  // Create log entry
  CreateLogMessagePara1 ( Timestamp   := AxesGroup.State.SystemTime,
                          MessageType := MessageType.CMD,
                          Severity    := Severity.ERROR,
                          MessageCode := ErrorID,
                          MessageText := 'Invalid Parameter ParCmd.JointPosition.E2 = {1}',
                          Para1       := VALID_REAL_TO_STRING(ParCmd.JointPosition.E2));
  RETURN;                          
END_IF


// Check ParCmd.JointPosition.E3 valid ? 
IF ( SysDepIsValidReal(ParCmd.JointPosition.E3) = FALSE ) 
THEN
  // Parameter not valid
  CheckParameterValid := FALSE;
  // Set error
  SetError( ErrorID := RobotLibraryErrorIdEnum.ERR_INVALID_PAR_CMD, Overwrite := TRUE );
  
  // Create log entry
  CreateLogMessagePara1 ( Timestamp   := AxesGroup.State.SystemTime,
                          MessageType := MessageType.CMD,
                          Severity    := Severity.ERROR,
                          MessageCode := ErrorID,
                          MessageText := 'Invalid Parameter ParCmd.JointPosition.E3 = {1}',
                          Para1       := VALID_REAL_TO_STRING(ParCmd.JointPosition.E3));
  RETURN;                          
END_IF


// Check ParCmd.JointPosition.E4 valid ? 
IF ( SysDepIsValidReal(ParCmd.JointPosition.E4) = FALSE ) 
THEN
  // Parameter not valid
  CheckParameterValid := FALSE;
  // Set error
  SetError( ErrorID := RobotLibraryErrorIdEnum.ERR_INVALID_PAR_CMD, Overwrite := TRUE );
  
  // Create log entry
  CreateLogMessagePara1 ( Timestamp   := AxesGroup.State.SystemTime,
                          MessageType := MessageType.CMD,
                          Severity    := Severity.ERROR,
                          MessageCode := ErrorID,
                          MessageText := 'Invalid Parameter ParCmd.JointPosition.E4 = {1}',
                          Para1       := VALID_REAL_TO_STRING(ParCmd.JointPosition.E4));
  RETURN;                          
END_IF


// Check ParCmd.JointPosition.E5 valid ? 
IF ( SysDepIsValidReal(ParCmd.JointPosition.E5) = FALSE ) 
THEN
  // Parameter not valid
  CheckParameterValid := FALSE;
  // Set error
  SetError( ErrorID := RobotLibraryErrorIdEnum.ERR_INVALID_PAR_CMD, Overwrite := TRUE );
  
  // Create log entry
  CreateLogMessagePara1 ( Timestamp   := AxesGroup.State.SystemTime,
                          MessageType := MessageType.CMD,
                          Severity    := Severity.ERROR,
                          MessageCode := ErrorID,
                          MessageText := 'Invalid Parameter ParCmd.JointPosition.E5 = {1}',
                          Para1       := VALID_REAL_TO_STRING(ParCmd.JointPosition.E5));
  RETURN;                          
END_IF


// Check ParCmd.JointPosition.E6 valid ? 
IF ( SysDepIsValidReal(ParCmd.JointPosition.E6) = FALSE ) 
THEN
  // Parameter not valid
  CheckParameterValid := FALSE;
  // Set error
  SetError( ErrorID := RobotLibraryErrorIdEnum.ERR_INVALID_PAR_CMD, Overwrite := TRUE );
  
  // Create log entry
  CreateLogMessagePara1 ( Timestamp   := AxesGroup.State.SystemTime,
                          MessageType := MessageType.CMD,
                          Severity    := Severity.ERROR,
                          MessageCode := ErrorID,
                          MessageText := 'Invalid Parameter ParCmd.JointPosition.E6 = {1}',
                          Para1       := VALID_REAL_TO_STRING(ParCmd.JointPosition.E6));
  RETURN;                          
END_IF


// Check ParCmd.DetectionMode valid ? 
IF (( ParCmd.DetectionMode <> DetectionMode.TORQUE             ) AND
    ( ParCmd.DetectionMode <> DetectionMode.FORCE              ) AND 
    ( ParCmd.DetectionMode <> DetectionMode.ELECTRICAL_CURRENT ) AND 
    ( ParCmd.DetectionMode <> DetectionMode.FOLLOWING_ERROR    ))  
THEN
  // Parameter not valid
  CheckParameterValid := FALSE;
  // Set error
  SetError( ErrorID := RobotLibraryErrorIdEnum.ERR_INVALID_PAR_CMD, Overwrite := TRUE );
  // Create log entry
  CreateLogMessagePara1 ( Timestamp   := AxesGroup.State.SystemTime,
                          MessageType := MessageType.CMD,
                          Severity    := Severity.ERROR,
                          MessageCode := ErrorID,
                          MessageText := 'Invalid Parameter ParCmd.DetectionMode = {1}',
                          Para1       := DETECTION_MODE_TO_STRING(ParCmd.DetectionMode));
  RETURN;                          
END_IF


FOR _idx := 0 TO 6
DO
  // Check ParCmd.DetectionVector[x] valid ? 
  IF ( SysDepIsValidReal(ParCmd.DetectionVector[_idx]) = FALSE ) 
  THEN
    // Parameter not valid
    CheckParameterValid := FALSE;
    // Set error
    SetError( ErrorID := RobotLibraryErrorIdEnum.ERR_INVALID_PAR_CMD, Overwrite := TRUE );
    
    // Create log entry
    CreateLogMessagePara2 ( Timestamp   := AxesGroup.State.SystemTime,
                            MessageType := MessageType.CMD,
                            Severity    := Severity.ERROR,
                            MessageCode := ErrorID,
                            MessageText := 'Invalid Parameter ParCmd.DetectionVector[{2}] = {1}',
                            Para1       := VALID_REAL_TO_STRING(ParCmd.DetectionVector[_idx]),
                            Para2       := DINT_TO_STRING(_idx));
    RETURN;                          
  END_IF
END_FOR


// Check ParCmd.VelocityRate valid ? 
IF  (( SysDepIsValidReal(ParCmd.VelocityRate) = FALSE )  OR
    ((                   ParCmd.VelocityRate  <     0 )  AND 
     (                   ParCmd.VelocityRate <>    -1 )) OR   
     (                   ParCmd.VelocityRate  >   100 ))      
THEN
  // Parameter not valid
  CheckParameterValid := FALSE;
  // Set error
  SetError( ErrorID := RobotLibraryErrorIdEnum.ERR_VELOCITY_INVALID, Overwrite := TRUE );
  // Create log entry
  CreateLogMessagePara1 ( Timestamp   := AxesGroup.State.SystemTime,
                          MessageType := MessageType.CMD,
                          Severity    := Severity.ERROR,
                          MessageCode := ErrorID,
                          MessageText := 'Invalid Parameter ParCmd.VelocityRate = {1}',
                          Para1       := VALID_REAL_TO_STRING(ParCmd.VelocityRate));                            
  RETURN;
END_IF


// Check ParCmd.AccelerationRate valid ? 
IF  (( SysDepIsValidReal(ParCmd.AccelerationRate) = FALSE )  OR
    ((                   ParCmd.AccelerationRate  <     0 )  AND 
     (                   ParCmd.AccelerationRate <>    -1 )) OR   
     (                   ParCmd.AccelerationRate  >   100 ))      
THEN
  // Parameter not valid
  CheckParameterValid := FALSE;
  // Set error
  SetError( ErrorID := RobotLibraryErrorIdEnum.ERR_ACCELERATION_INVALID, Overwrite := TRUE );
  // Create log entry
  CreateLogMessagePara1 ( Timestamp   := AxesGroup.State.SystemTime,
                          MessageType := MessageType.CMD,
                          Severity    := Severity.ERROR,
                          MessageCode := ErrorID,
                          MessageText := 'Invalid Parameter ParCmd.AccelerationRate = {1}',
                          Para1       := VALID_REAL_TO_STRING(ParCmd.AccelerationRate));                            
  RETURN;
END_IF


// Check ParCmd.DecelerationRate valid ? 
IF  (( SysDepIsValidReal(ParCmd.DecelerationRate) = FALSE )  OR
    ((                   ParCmd.DecelerationRate  <     0 )  AND 
     (                   ParCmd.DecelerationRate <>    -1 )) OR   
     (                   ParCmd.DecelerationRate  >   100 ))      
THEN
  // Parameter not valid
  CheckParameterValid := FALSE;
  // Set error
  SetError( ErrorID := RobotLibraryErrorIdEnum.ERR_DECELERATION_INVALID, Overwrite := TRUE );
  // Create log entry
  CreateLogMessagePara1 ( Timestamp   := AxesGroup.State.SystemTime,
                          MessageType := MessageType.CMD,
                          Severity    := Severity.ERROR,
                          MessageCode := ErrorID,
                          MessageText := 'Invalid Parameter ParCmd.DecelerationRate = {1}',
                          Para1       := VALID_REAL_TO_STRING(ParCmd.DecelerationRate));                            
  RETURN;
END_IF


// Check ParCmd.JerkRate valid ? 
IF  (( SysDepIsValidReal(ParCmd.JerkRate) = FALSE )  OR
    ((                   ParCmd.JerkRate  <     0 )  AND 
     (                   ParCmd.JerkRate <>    -1 )) OR   
     (                   ParCmd.JerkRate  >   100 ))      
THEN
  // Parameter not valid
  CheckParameterValid := FALSE;
  // Set error
  SetError( ErrorID := RobotLibraryErrorIdEnum.ERR_JERK_INVALID, Overwrite := TRUE );
  // Create log entry
  CreateLogMessagePara1 ( Timestamp   := AxesGroup.State.SystemTime,
                          MessageType := MessageType.CMD,
                          Severity    := Severity.ERROR,
                          MessageCode := ErrorID,
                          MessageText := 'Invalid Parameter ParCmd.JerkRate = {1}',
                          Para1       := VALID_REAL_TO_STRING(ParCmd.JerkRate));                            
  RETURN;
END_IF


// Check ParCmd.Manipulation
// -> no plausibility check for boolean
                
END_METHOD

METHOD INTERNAL CreateCommandPayload : RobotLibraryCommandDataFB
VAR_IN_OUT
  /// Robot assignment of function
  AxesGroup : AxesGroup; 
END_VAR
VAR
  /// Parameter count
 _parameterCnt : DINT;
END_VAR
// Table 6-412: Sent CMD payload (PLC to RC) of "SearchHardStopJ"
// --------------------------
// Header
// --------------------------
// Byte 00 : UINT  - Type HB     
// Byte 01 :       - Type LB    
// Byte 02 : USINT - Reserve | ExecutionMode
// Byte 03 : USINT - ParSeq  | Priority
// --------------------------
// Datablock
// --------------------------
// Byte 04 : UINT  VelocityRate;
// Byte 05 :       VelocityRate;
// Byte 06 : UINT  AccelerationRate;
// Byte 07 :       AccelerationRate;
// Byte 08 : UINT  DecelerationRate;
// Byte 09 :       DecelerationRate;
// Byte 10 : UINT  JerkRate;
// Byte 11 :       JerkRate;
// Byte 12 : REAL  JointPosition.J1;
// Byte 13 :       JointPosition.J1;
// Byte 14 :       JointPosition.J1;
// Byte 15 :       JointPosition.J1;
// Byte 16 : REAL  JointPosition.J2;
// Byte 17 :       JointPosition.J2;
// Byte 18 :       JointPosition.J2;
// Byte 19 :       JointPosition.J2;
// Byte 20 : REAL  JointPosition.J3;
// Byte 21 :       JointPosition.J3;
// Byte 22 :       JointPosition.J3;
// Byte 23 :       JointPosition.J3;
// Byte 24 : REAL  JointPosition.J4;
// Byte 25 :       JointPosition.J4;
// Byte 26 :       JointPosition.J4;
// Byte 27 :       JointPosition.J4;
// Byte 28 : REAL  JointPosition.J5;
// Byte 29 :       JointPosition.J5;
// Byte 30 :       JointPosition.J5;
// Byte 31 :       JointPosition.J5;
// Byte 32 : REAL  JointPosition.J6;
// Byte 33 :       JointPosition.J6;
// Byte 34 :       JointPosition.J6;
// Byte 35 :       JointPosition.J6;
// Byte 36 : REAL  JointPosition.E1;
// Byte 37 :       JointPosition.E1;
// Byte 38 :       JointPosition.E1;
// Byte 39 :       JointPosition.E1;
// Byte 40 : USINT OriMode;
// Byte 41 : USINT DetectionMode;
// Byte 42 : BOOL  Manipulation;
// Byte 43 : BYTE  Reserved;
// Byte 44 : REAL  DetectionVector[0];
// Byte 45 :       DetectionVector[0];
// Byte 46 :       DetectionVector[0];
// Byte 47 :       DetectionVector[0];
// Byte 48 : REAL  DetectionVector[1];
// Byte 49 :       DetectionVector[1];
// Byte 50 :       DetectionVector[1];
// Byte 51 :       DetectionVector[1];
// Byte 52 : REAL  DetectionVector[2];
// Byte 53 :       DetectionVector[2];
// Byte 54 :       DetectionVector[2];
// Byte 55 :       DetectionVector[2];
// Byte 56 : REAL  DetectionVector[3];
// Byte 57 :       DetectionVector[3];
// Byte 58 :       DetectionVector[3];
// Byte 59 :       DetectionVector[3];
// Byte 60 : REAL  DetectionVector[4];
// Byte 61 :       DetectionVector[4];
// Byte 62 :       DetectionVector[4];
// Byte 63 :       DetectionVector[4];
// Byte 64 : REAL  DetectionVector[5];
// Byte 65 :       DetectionVector[5];
// Byte 66 :       DetectionVector[5];
// Byte 67 :       DetectionVector[5];
// Byte 68 : REAL  JointPosition.E2;
// Byte 69 :       JointPosition.E2;
// Byte 70 :       JointPosition.E2;
// Byte 71 :       JointPosition.E2;
// Byte 72 : REAL  JointPosition.E3;
// Byte 73 :       JointPosition.E3;
// Byte 74 :       JointPosition.E3;
// Byte 75 :       JointPosition.E3;
// Byte 76 : REAL  JointPosition.E4;
// Byte 77 :       JointPosition.E4;
// Byte 78 :       JointPosition.E4;
// Byte 79 :       JointPosition.E4;
// Byte 80 : REAL  JointPosition.E5;
// Byte 81 :       JointPosition.E5;
// Byte 82 :       JointPosition.E5;
// Byte 83 :       JointPosition.E5;
// Byte 84 : REAL  JointPosition.E6;
// Byte 85 :       JointPosition.E6;
// Byte 86 :       JointPosition.E6;
// Byte 87 :       JointPosition.E6;
// --------------------------
                  // set command parameter 
_command.CmdTyp            :=  CmdType.SearchHardstopJ;
_command.ExecMode          :=  ExecMode;
_command.ParSeq            := _command.ParSeq;
_command.Priority          :=  Priority;
_command.VelocityRate      :=  REAL_TO_PERCENT_UINT(_parCmd.VelocityRate     , IsOptional := FALSE);
_command.AccelerationRate  :=  REAL_TO_PERCENT_UINT(_parCmd.AccelerationRate , IsOptional := FALSE);
_command.DecelerationRate  :=  REAL_TO_PERCENT_UINT(_parCmd.DecelerationRate , IsOptional := TRUE );
_command.JerkRate          :=  REAL_TO_PERCENT_UINT(_parCmd.JerkRate         , IsOptional := TRUE );
_command.JointPosition     := _parCmd.JointPosition;
_command.OriMode           := 0;
_command.DetectionMode     := _parCmd.DetectionMode;
_command.Manipulation      := _parCmd.Manipulation;
_command.Reserve           :=  0;
_command.DetectionVector   := _parCmd.DetectionVector;

// copy command data to header
_cmdHeader := _command;
// call base implementation to copy header to payload buffer
CreateCommandPayload := SUPER^.CreateCommandPayload(AxesGroup := AxesGroup);


// Check parameter must be added ? 
IF ( CheckAddParameter(CreateCommandPayload.PayloadPtr))
THEN
  // add command.VelocityRate
  CreateCommandPayload.AddUint(_command.VelocityRate);
  // inc parameter counter
 _parameterCnt := _parameterCnt + 1;  
END_IF

// Check parameter must be added ? 
IF ( CheckAddParameter(CreateCommandPayload.PayloadPtr))
THEN
  // add command.AccelerationRate
  CreateCommandPayload.AddUint(_command.AccelerationRate);
  // inc parameter counter
 _parameterCnt := _parameterCnt + 1;  
END_IF


// Check parameter must be added ? 
IF ( CheckAddParameter(CreateCommandPayload.PayloadPtr))
THEN
  // add command.DecelerationRate
  CreateCommandPayload.AddUint(_command.DecelerationRate);
  // inc parameter counter
 _parameterCnt := _parameterCnt + 1;  
END_IF


// Check parameter must be added ? 
IF ( CheckAddParameter(CreateCommandPayload.PayloadPtr))
THEN
  // add command.JerkRate
  CreateCommandPayload.AddUint(_command.JerkRate);
  // inc parameter counter
 _parameterCnt := _parameterCnt + 1;  
END_IF


// Check parameter must be added ? 
IF ( CheckAddParameter(CreateCommandPayload.PayloadPtr))
THEN
  // add command.JointPosition.J1
  CreateCommandPayload.AddReal(_command.JointPosition.J1);
  // inc parameter counter
 _parameterCnt := _parameterCnt + 1;  
END_IF


// Check parameter must be added ? 
IF ( CheckAddParameter(CreateCommandPayload.PayloadPtr))
THEN
  // add command.JointPosition.J2
  CreateCommandPayload.AddReal(_command.JointPosition.J2);
  // inc parameter counter
 _parameterCnt := _parameterCnt + 1;  
END_IF


// Check parameter must be added ? 
IF ( CheckAddParameter(CreateCommandPayload.PayloadPtr))
THEN
  // add command.JointPosition.J3
  CreateCommandPayload.AddReal(_command.JointPosition.J3);
  // inc parameter counter
 _parameterCnt := _parameterCnt + 1;  
END_IF


// Check parameter must be added ? 
IF ( CheckAddParameter(CreateCommandPayload.PayloadPtr))
THEN
  // add command.JointPosition.J4
  CreateCommandPayload.AddReal(_command.JointPosition.J4);
  // inc parameter counter
 _parameterCnt := _parameterCnt + 1;  
END_IF


// Check parameter must be added ? 
IF ( CheckAddParameter(CreateCommandPayload.PayloadPtr))
THEN
  // add command.JointPosition.J5
  CreateCommandPayload.AddReal(_command.JointPosition.J5);
  // inc parameter counter
 _parameterCnt := _parameterCnt + 1;  
END_IF


// Check parameter must be added ? 
IF ( CheckAddParameter(CreateCommandPayload.PayloadPtr))
THEN
  // add command.JointPosition.J6
  CreateCommandPayload.AddReal(_command.JointPosition.J6);
  // inc parameter counter
 _parameterCnt := _parameterCnt + 1;  
END_IF


// Check parameter must be added ? 
IF ( CheckAddParameter(CreateCommandPayload.PayloadPtr))
THEN
  // add command.JointPosition.E1
  CreateCommandPayload.AddReal(_command.JointPosition.E1);
  // inc parameter counter
 _parameterCnt := _parameterCnt + 1;  
END_IF


// Check parameter must be added ? 
IF ( CheckAddParameter(CreateCommandPayload.PayloadPtr))
THEN
  // add command.OriMode
  CreateCommandPayload.AddUsint(_command.OriMode);
  // inc parameter counter
 _parameterCnt := _parameterCnt + 1;  
END_IF


// Check parameter must be added ? 
IF ( CheckAddParameter(CreateCommandPayload.PayloadPtr))
THEN
  // add command.DetectionMode
  CreateCommandPayload.AddUsint(_command.DetectionMode);
  // inc parameter counter
 _parameterCnt := _parameterCnt + 1;  
END_IF


// Check parameter must be added ? 
IF ( CheckAddParameter(CreateCommandPayload.PayloadPtr))
THEN
  // add command.Manipulation
  CreateCommandPayload.AddBool(_command.Manipulation);
  // inc parameter counter
 _parameterCnt := _parameterCnt + 1;  
END_IF


// Check parameter must be added ? 
IF ( CheckAddParameter(CreateCommandPayload.PayloadPtr))
THEN
  // add command.Reserve
  CreateCommandPayload.AddByte(_command.Reserve);
  // inc parameter counter
 _parameterCnt := _parameterCnt + 1;  
END_IF


// Check parameter must be added ? 
IF ( CheckAddParameter(CreateCommandPayload.PayloadPtr))
THEN
  // add command.DetectionVector[0]
  CreateCommandPayload.AddReal(_command.DetectionVector[0]);
  // inc parameter counter
 _parameterCnt := _parameterCnt + 1;  
END_IF


// Check parameter must be added ? 
IF ( CheckAddParameter(CreateCommandPayload.PayloadPtr))
THEN
  // add command.DetectionVector[1]
  CreateCommandPayload.AddReal(_command.DetectionVector[1]);
  // inc parameter counter
 _parameterCnt := _parameterCnt + 1;  
END_IF


// Check parameter must be added ? 
IF ( CheckAddParameter(CreateCommandPayload.PayloadPtr))
THEN
  // add command.DetectionVector[2]
  CreateCommandPayload.AddReal(_command.DetectionVector[2]);
  // inc parameter counter
 _parameterCnt := _parameterCnt + 1;  
END_IF


// Check parameter must be added ? 
IF ( CheckAddParameter(CreateCommandPayload.PayloadPtr))
THEN
  // add command.DetectionVector[3]
  CreateCommandPayload.AddReal(_command.DetectionVector[3]);
  // inc parameter counter
 _parameterCnt := _parameterCnt + 1;  
END_IF


// Check parameter must be added ? 
IF ( CheckAddParameter(CreateCommandPayload.PayloadPtr))
THEN
  // add command.DetectionVector[4]
  CreateCommandPayload.AddReal(_command.DetectionVector[4]);
  // inc parameter counter
 _parameterCnt := _parameterCnt + 1;  
END_IF


// Check parameter must be added ? 
IF ( CheckAddParameter(CreateCommandPayload.PayloadPtr))
THEN
  // add command.DetectionVector[5]
  CreateCommandPayload.AddReal(_command.DetectionVector[5]);
  // inc parameter counter
 _parameterCnt := _parameterCnt + 1;  
END_IF


// Check parameter must be added ? 
IF ( CheckAddParameter(CreateCommandPayload.PayloadPtr))
THEN
  // add command.JointPosition.E2
  CreateCommandPayload.AddReal(_command.JointPosition.E2);
  // inc parameter counter
 _parameterCnt := _parameterCnt + 1;  
END_IF


// Check parameter must be added ? 
IF ( CheckAddParameter(CreateCommandPayload.PayloadPtr))
THEN
  // add command.JointPosition.E3
  CreateCommandPayload.AddReal(_command.JointPosition.E3);
  // inc parameter counter
 _parameterCnt := _parameterCnt + 1;  
END_IF


// Check parameter must be added ? 
IF ( CheckAddParameter(CreateCommandPayload.PayloadPtr))
THEN
  // add command.JointPosition.E4
  CreateCommandPayload.AddReal(_command.JointPosition.E4);
  // inc parameter counter
 _parameterCnt := _parameterCnt + 1;  
END_IF


// Check parameter must be added ? 
IF ( CheckAddParameter(CreateCommandPayload.PayloadPtr))
THEN
  // add command.JointPosition.E5
  CreateCommandPayload.AddReal(_command.JointPosition.E5);
  // inc parameter counter
 _parameterCnt := _parameterCnt + 1;  
END_IF


// Check parameter must be added ? 
IF ( CheckAddParameter(CreateCommandPayload.PayloadPtr))
THEN
  // add command.JointPosition.E6
  CreateCommandPayload.AddReal(_command.JointPosition.E6);
  // inc parameter counter
 _parameterCnt := _parameterCnt + 1;  
END_IF

  
// Create logging
CreateCommandPayloadLog(AxesGroup := AxesGroup, ParameterCnt := _parameterCnt);
                
END_METHOD

METHOD INTERNAL CreateCommandPayloadLog
VAR_IN_OUT
  /// Robot assignment of function
  AxesGroup : AxesGroup; 
END_VAR
VAR_INPUT
  /// Parameter count
  ParameterCnt : DINT;
END_VAR
VAR 
  /// internal index for loops
 _idx : DINT;
END_VAR
                  // Create log entry for Parameter start
CreateLogMessagePara1 ( Timestamp   := AxesGroup.State.SystemTime,
                        MessageType := MessageType.CMD,
                        Severity    := Severity.DEBUG,
                        MessageCode := 0,
                        MessageText := 'Create command payload with {1} parameter(s) :',
                        Para1       := DINT_TO_STRING(ParameterCnt));
  

// Return if no parameter is remaining...
IF ( ParameterCnt = 0 ) THEN RETURN; END_IF
// dec remaining parameter(s)                        
ParameterCnt := ParameterCnt - 1;
// Create log entry for VelocityRate
CreateLogMessagePara1 ( Timestamp   := AxesGroup.State.SystemTime,
                        MessageType := MessageType.CMD,
                        Severity    := Severity.DEBUG,
                        MessageCode := 0,
                        MessageText := 'Command.VelocityRate = {1}',
                        Para1       :=  UINT_TO_STRING(_command.VelocityRate));


// Return if no parameter is remaining...
IF ( ParameterCnt = 0 ) THEN RETURN; END_IF
// dec remaining parameter(s)                        
ParameterCnt := ParameterCnt - 1;
// Create log entry for AccelerationRate
CreateLogMessagePara1 ( Timestamp   := AxesGroup.State.SystemTime,
                        MessageType := MessageType.CMD,
                        Severity    := Severity.DEBUG,
                        MessageCode := 0,
                        MessageText := 'Command.AccelerationRate = {1}',
                        Para1       :=  UINT_TO_STRING(_command.AccelerationRate));
                        

// Return if no parameter is remaining...
IF ( ParameterCnt = 0 ) THEN RETURN; END_IF
// dec remaining parameter(s)                        
ParameterCnt := ParameterCnt - 1;
// Create log entry for DecelerationRate
CreateLogMessagePara1 ( Timestamp   := AxesGroup.State.SystemTime,
                        MessageType := MessageType.CMD,
                        Severity    := Severity.DEBUG,
                        MessageCode := 0,
                        MessageText := 'Command.DecelerationRate = {1}',
                        Para1       :=  UINT_TO_STRING(_command.DecelerationRate));


// Return if no parameter is remaining...
IF ( ParameterCnt = 0 ) THEN RETURN; END_IF
// dec remaining parameter(s)                        
ParameterCnt := ParameterCnt - 1;
// Create log entry for JerkRate
CreateLogMessagePara1 ( Timestamp   := AxesGroup.State.SystemTime,
                        MessageType := MessageType.CMD,
                        Severity    := Severity.DEBUG,
                        MessageCode := 0,
                        MessageText := 'Command.JerkRate = {1}',
                        Para1       :=  UINT_TO_STRING(_command.JerkRate));


// Return if no parameter is remaining...
IF ( ParameterCnt = 0 ) THEN RETURN; END_IF
// dec remaining parameter(s)                        
ParameterCnt := ParameterCnt - 1;
// Create log entry for JointPosition.J1
CreateLogMessagePara1 ( Timestamp   := AxesGroup.State.SystemTime,
                        MessageType := MessageType.CMD,
                        Severity    := Severity.DEBUG,
                        MessageCode := 0,
                        MessageText := 'Command.JointPosition.J1 = {1}',
                        Para1       :=  REAL_TO_STRING(_command.JointPosition.J1));


// Return if no parameter is remaining...
IF ( ParameterCnt = 0 ) THEN RETURN; END_IF
// dec remaining parameter(s)                        
ParameterCnt := ParameterCnt - 1;
// Create log entry for JointPosition.J2
CreateLogMessagePara1 ( Timestamp   := AxesGroup.State.SystemTime,
                        MessageType := MessageType.CMD,
                        Severity    := Severity.DEBUG,
                        MessageCode := 0,
                        MessageText := 'Command.JointPosition.J2 = {1}',
                        Para1       :=  REAL_TO_STRING(_command.JointPosition.J2));


// Return if no parameter is remaining...
IF ( ParameterCnt = 0 ) THEN RETURN; END_IF
// dec remaining parameter(s)                        
ParameterCnt := ParameterCnt - 1;
// Create log entry for JointPosition.J3
CreateLogMessagePara1 ( Timestamp   := AxesGroup.State.SystemTime,
                        MessageType := MessageType.CMD,
                        Severity    := Severity.DEBUG,
                        MessageCode := 0,
                        MessageText := 'Command.JointPosition.J3 = {1}',
                        Para1       :=  REAL_TO_STRING(_command.JointPosition.J3));


// Return if no parameter is remaining...
IF ( ParameterCnt = 0 ) THEN RETURN; END_IF
// dec remaining parameter(s)                        
ParameterCnt := ParameterCnt - 1;
// Create log entry for JointPosition.J4
CreateLogMessagePara1 ( Timestamp   := AxesGroup.State.SystemTime,
                        MessageType := MessageType.CMD,
                        Severity    := Severity.DEBUG,
                        MessageCode := 0,
                        MessageText := 'Command.JointPosition.J4 = {1}',
                        Para1       :=  REAL_TO_STRING(_command.JointPosition.J4));


// Return if no parameter is remaining...
IF ( ParameterCnt = 0 ) THEN RETURN; END_IF
// dec remaining parameter(s)                        
ParameterCnt := ParameterCnt - 1;
// Create log entry for JointPosition.J5
CreateLogMessagePara1 ( Timestamp   := AxesGroup.State.SystemTime,
                        MessageType := MessageType.CMD,
                        Severity    := Severity.DEBUG,
                        MessageCode := 0,
                        MessageText := 'Command.JointPosition.J5 = {1}',
                        Para1       :=  REAL_TO_STRING(_command.JointPosition.J5));


// Return if no parameter is remaining...
IF ( ParameterCnt = 0 ) THEN RETURN; END_IF
// dec remaining parameter(s)                        
ParameterCnt := ParameterCnt - 1;
// Create log entry for JointPosition.J6
CreateLogMessagePara1 ( Timestamp   := AxesGroup.State.SystemTime,
                        MessageType := MessageType.CMD,
                        Severity    := Severity.DEBUG,
                        MessageCode := 0,
                        MessageText := 'Command.JointPosition.J6 = {1}',
                        Para1       :=  REAL_TO_STRING(_command.JointPosition.J6));


// Return if no parameter is remaining...
IF ( ParameterCnt = 0 ) THEN RETURN; END_IF
// dec remaining parameter(s)                        
ParameterCnt := ParameterCnt - 1;
// Create log entry for JointPosition.E1
CreateLogMessagePara1 ( Timestamp   := AxesGroup.State.SystemTime,
                        MessageType := MessageType.CMD,
                        Severity    := Severity.DEBUG,
                        MessageCode := 0,
                        MessageText := 'Command.JointPosition.E1 = {1}',
                        Para1       :=  REAL_TO_STRING(_command.JointPosition.E1));


// Return if no parameter is remaining...
IF ( ParameterCnt = 0 ) THEN RETURN; END_IF
// dec remaining parameter(s)                        
ParameterCnt := ParameterCnt - 1;
// Create log entry for OriMode
CreateLogMessagePara1 ( Timestamp   := AxesGroup.State.SystemTime,
                        MessageType := MessageType.CMD,
                        Severity    := Severity.DEBUG,
                        MessageCode := 0,
                        MessageText := 'Command.OriMode = {1}',
                        Para1       :=  ORI_MODE_TO_STRING(_command.OriMode));


// Return if no parameter is remaining...
IF ( ParameterCnt = 0 ) THEN RETURN; END_IF
// dec remaining parameter(s)                        
ParameterCnt := ParameterCnt - 1;
// Create log entry for DetectionMode
CreateLogMessagePara1 ( Timestamp   := AxesGroup.State.SystemTime,
                        MessageType := MessageType.CMD,
                        Severity    := Severity.DEBUG,
                        MessageCode := 0,
                        MessageText := 'Command.DetectionMode = {1}',
                        Para1       :=  DETECTION_MODE_TO_STRING(_command.DetectionMode));


// Return if no parameter is remaining...
IF ( ParameterCnt = 0 ) THEN RETURN; END_IF
// dec remaining parameter(s)                        
ParameterCnt := ParameterCnt - 1;
// Create log entry for Manipulation
CreateLogMessagePara1 ( Timestamp   := AxesGroup.State.SystemTime,
                        MessageType := MessageType.CMD,
                        Severity    := Severity.DEBUG,
                        MessageCode := 0,
                        MessageText := 'Command.Manipulation = {1}',
                        Para1       :=  BOOL_TO_STRING(_command.Manipulation));


// Return if no parameter is remaining...
IF ( ParameterCnt = 0 ) THEN RETURN; END_IF
// dec remaining parameter(s)                        
ParameterCnt := ParameterCnt - 1;
// Create log entry for Reserve
CreateLogMessagePara1 ( Timestamp   := AxesGroup.State.SystemTime,
                        MessageType := MessageType.CMD,
                        Severity    := Severity.DEBUG,
                        MessageCode := 0,
                        MessageText := 'Command.Reserve = {1}',
                        Para1       :=  USINT_TO_STRING(_command.Reserve));


// Create log entry for DetectionVector[x]
FOR _idx := 0 TO 5
DO
  // Return if no parameter is remaining...
  IF ( ParameterCnt = 0 ) THEN RETURN; END_IF
  // dec remaining parameter(s)                        
  ParameterCnt := ParameterCnt - 1;
  // Create log entry for Commmand.DetectionVector
  CreateLogMessagePara2 ( Timestamp   := AxesGroup.State.SystemTime,
                          MessageType := MessageType.CMD,
                          Severity    := Severity.DEBUG,
                          MessageCode := 0,
                          MessageText := 'Command.DetectionVector[{2}] = {1}',
                          Para1       :=  REAL_TO_STRING(_command.DetectionVector[_idx]),
                          Para2       :=  DINT_TO_STRING(_idx));
END_FOR


// Return if no parameter is remaining...
IF ( ParameterCnt = 0 ) THEN RETURN; END_IF
// dec remaining parameter(s)                        
ParameterCnt := ParameterCnt - 1;
// Create log entry for JointPosition.E2
CreateLogMessagePara1 ( Timestamp   := AxesGroup.State.SystemTime,
                        MessageType := MessageType.CMD,
                        Severity    := Severity.DEBUG,
                        MessageCode := 0,
                        MessageText := 'Command.JointPosition.E2 = {1}',
                        Para1       :=  REAL_TO_STRING(_command.JointPosition.E2));


// Return if no parameter is remaining...
IF ( ParameterCnt = 0 ) THEN RETURN; END_IF
// dec remaining parameter(s)                        
ParameterCnt := ParameterCnt - 1;
// Create log entry for JointPosition.E3
CreateLogMessagePara1 ( Timestamp   := AxesGroup.State.SystemTime,
                        MessageType := MessageType.CMD,
                        Severity    := Severity.DEBUG,
                        MessageCode := 0,
                        MessageText := 'Command.JointPosition.E3 = {1}',
                        Para1       :=  REAL_TO_STRING(_command.JointPosition.E3));


// Return if no parameter is remaining...
IF ( ParameterCnt = 0 ) THEN RETURN; END_IF
// dec remaining parameter(s)                        
ParameterCnt := ParameterCnt - 1;
// Create log entry for JointPosition.E4
CreateLogMessagePara1 ( Timestamp   := AxesGroup.State.SystemTime,
                        MessageType := MessageType.CMD,
                        Severity    := Severity.DEBUG,
                        MessageCode := 0,
                        MessageText := 'Command.JointPosition.E4 = {1}',
                        Para1       :=  REAL_TO_STRING(_command.JointPosition.E4));


// Return if no parameter is remaining...
IF ( ParameterCnt = 0 ) THEN RETURN; END_IF
// dec remaining parameter(s)                        
ParameterCnt := ParameterCnt - 1;
// Create log entry for JointPosition.E5
CreateLogMessagePara1 ( Timestamp   := AxesGroup.State.SystemTime,
                        MessageType := MessageType.CMD,
                        Severity    := Severity.DEBUG,
                        MessageCode := 0,
                        MessageText := 'Command.JointPosition.E5 = {1}',
                        Para1       :=  REAL_TO_STRING(_command.JointPosition.E5));


// Return if no parameter is remaining...
IF ( ParameterCnt = 0 ) THEN RETURN; END_IF
// dec remaining parameter(s)                        
ParameterCnt := ParameterCnt - 1;
// Create log entry for JointPosition.E6
CreateLogMessagePara1 ( Timestamp   := AxesGroup.State.SystemTime,
                        MessageType := MessageType.CMD,
                        Severity    := Severity.DEBUG,
                        MessageCode := 0,
                        MessageText := 'Command.JointPosition.E6 = {1}',
                        Para1       :=  REAL_TO_STRING(_command.JointPosition.E6));
                
END_METHOD

METHOD FB_init : BOOL
VAR_INPUT
  /// if TRUE, the retain variables are initialized (warm start / cold start)
  bInitRetains : BOOL; 
  /// if TRUE, the instance afterwards gets moved into the copy code (online change)
  bInCopyCode  : BOOL;  
END_VAR
                  MyType := 'MC_SearchHardStopJFB';

ExecMode     := ExecutionMode.SEQUENCE_PRIMARY;
Priority     := PriorityLevel.NORMAL;
SequenceFlag := SequenceFlagEnum.PRIMARY_SEQUENCE;  

                
END_METHOD

METHOD PROTECTED OnApplyOutCmd
VAR_INPUT
  /// Command message state
  State : CmdMessageState;
END_VAR
                  IF ( State = CmdMessageState.EMPTY ) 
THEN
  // Reset command outputs
  SysDepMemSet(pDest := ADR(OutCmd), Value := 0, DataLen := SIZEOF(OutCmd));         
END_IF

IF (( State = CmdMessageState.ACTIVE ) OR
    ( State = CmdMessageState.DONE   ))
THEN
  // Update results
  OutCmd.InClamping        := _response.InClamping;
  OutCmd.Progress          :=  PERCENT_UINT_TO_REAL( Value := _response.Progress, IsOptional := TRUE);
  OutCmd.RemainingDistance := _response.RemainingDistance;
END_IF
                
END_METHOD

METHOD PROTECTED OnExecRun : DINT
VAR_IN_OUT
  /// Robot assignment of function
  AxesGroup : AxesGroup; 
END_VAR
                  // call base implementation
SUPER^.OnExecRun(AxesGroup := AxesGroup);

CASE _stepCmd OF
  
  00:  IF ( _execute_R.Q ) AND ( NOT Error)  
       THEN
         // Check function is supported and parameter are valid ?
         IF (( CheckFunctionSupported( AxesGroup := AxesGroup )) AND
             ( CheckParameterValid   ( AxesGroup := AxesGroup )))
         THEN      
           // set busy flag
           Busy := TRUE;
           // Reset command outputs
           SysDepMemSet(pDest := ADR(OutCmd), Value := 0, DataLen := SIZEOF(OutCmd));         
           // apply command parameter
          _parCmd := ParCmd;
           // init parameter sequence
          _command.ParSeq := 1;
           // create command data
           CommandData := CreateCommandPayload(AxesGroup := AxesGroup);
           // Add command to active command register
          _uniqueID := AxesGroup.Acyclic.ActiveCommandRegister.AddCmd( pCommandFB := ADR(THIS^ ));     
           // set timeout
           SetTimeout(PT := _timeoutCmd, rTimer := _timerCmd);
           // inc step counter
          _stepCmd := _stepCmd + 1;
         END_IF 
       END_IF
     

  01:  // Wait for responce received
       IF ( _responseReceived )
       THEN
         // reset response received flag
        _responseReceived := FALSE;
         // update state flags
         OnUpdateStateFlags(_response.State);
         // update state flags
         OnApplyOutCmd(_response.State);
                
         // Done, Aborted or Error ?
         IF (_response.State >= CmdMessageState.DONE )
         THEN
           // set timeout
           SetTimeout(PT := _timeoutCmd, rTimer := _timerCmd);
           // inc step counter
          _stepCmd := _stepCmd + 1; 
         END_IF
       END_IF


  02: IF ( NOT Execute)
      THEN
        Reset();  
      END_IF     

ELSE
  // invalid step
  SetError( ErrorID := RobotLibraryErrorIdEnum.ERR_INVALID_STEP, Overwrite := TRUE );
END_CASE


// Reset FB
IF ( NOT Execute )
THEN
  Reset();  
END_IF
                
END_METHOD

METHOD PROTECTED OnUpdateStateFlags
VAR_INPUT
  /// Command message state
  State : CmdMessageState;
END_VAR
                  // Reset State flags
Active             := FALSE;
CommandAborted     := FALSE;
CommandInterrupted := FALSE;
Done               := FALSE;

CASE State OF

  // No operation or process is active
  CmdMessageState.EMPTY               :;
  // Created but not yet started
  CmdMessageState.CREATED             :;
  // Buffered and awaiting execution
  CmdMessageState.BUFFERED            : CommandBuffered    := TRUE;
  // Buffered in planner for future execution
  CmdMessageState.BUFFERED_IN_PLANNER : CommandBuffered    := TRUE;
  // Currently active and in progress
  CmdMessageState.ACTIVE              : Active             := TRUE;                                   
  // Interrupted and awaiting continuation
  CmdMessageState.INTERRUPTED         : CommandInterrupted := TRUE;     
  // Requested for abort
  CmdMessageState.ABORT_REQUEST       :;
  // Successfully completed
  CmdMessageState.DONE                : Done               := TRUE; 
                                        Busy               := FALSE;
  // Aborted before completion
  CmdMessageState.ABORTED             : CommandAborted     := TRUE;
                                        Busy               := FALSE;
  // Encountered an error during execution
  CmdMessageState.ERROR               : Error              := TRUE;
                                        Busy               := FALSE;
END_CASE
                
END_METHOD

METHOD INTERNAL ParseResponsePayload : DINT
VAR_INPUT
  /// Response data
  ResponseData : RobotLibraryResponseDataFB;
  /// Timestamp
  Timestamp    : SystemTime;  
END_VAR
VAR
  /// Parameter count
 _parameterCnt : DINT;
END_VAR
// Table 6-413: Received CMD payload (RC to PLC) of "SearchHardStopJ"
// --------------------------
// Header
// --------------------------
// Byte 00 : USINT   - ParSeq | State     
// Byte 01 : SINT    - AlarmMessageSeverity    
// Byte 02 : UINT    - AlarmMessageCode HB
// Byte 03 :         - AlarmMessageCode LB
// --------------------------
// Datablock
// --------------------------
// Byte 04 : UINT    - Progress LW HB
// Byte 05 :         - Progress LW LB
// Byte 06 : REAL    - RemainingDistance HW HB
// Byte 07 :         - RemainingDistance HW LB
// Byte 08 :         - RemainingDistance LW HB
// Byte 09 :         - RemainingDistance LW LB
// Byte 10 : BOOL    - InClamping
                  // call base implementation to parse the header from payload buffer
ResponseData.PayloadPtr := SUPER^.ParseResponsePayload(ResponseData := ResponseData, Timestamp := Timestamp);

// copy parsed header to response
_response.ParSeq               := _rspHeader.ParSeq;
_response.State                := _rspHeader.State;
_response.AlarmMessageSeverity := _rspHeader.AlarmMessageSeverity;
_response.AlarmMessageCode     := _rspHeader.AlarmMessageCode;


// Check payload remaining ? 
IF ( ResponseData.IsPayloadRemaining)
THEN  
  // Get Response.Progress
 _response.Progress := ResponseData.GetUint();
  // inc parameter counter
 _parameterCnt := _parameterCnt + 1;
END_IF


// Check payload remaining ? 
IF ( ResponseData.IsPayloadRemaining)
THEN  
  // Get Response.RemainingDistance
 _response.RemainingDistance := ResponseData.GetReal();
  // inc parameter counter
 _parameterCnt := _parameterCnt + 1;
END_IF


// Check payload remaining ? 
IF ( ResponseData.IsPayloadRemaining)
THEN  
  // Get Response.InClamping
 _response.InClamping := ResponseData.GetBool();
  // inc parameter counter
 _parameterCnt := _parameterCnt + 1;
END_IF

 
// Create logging
ParseResponsePayloadLog(ResponseData := ResponseData, Timestamp := Timestamp, ParameterCnt := _parameterCnt);
                
END_METHOD

METHOD INTERNAL ParseResponsePayloadLog
VAR_INPUT
  /// Response data
  ResponseData : RobotLibraryResponseDataFB;
  /// Timestamp
  Timestamp    : SystemTime;  
  /// Parameter count
  ParameterCnt : DINT;
END_VAR
                  // Create log entry for Parameter start
CreateLogMessagePara1 ( Timestamp   := Timestamp,
                        MessageType := MessageType.CMD,
                        Severity    := Severity.DEBUG,
                        MessageCode := 0,
                        MessageText := '{1} parameter(s) to parse from the response data:',
                        Para1       := DINT_TO_STRING(ParameterCnt));
                        

// Return if no parameter is remaining...
IF ( ParameterCnt = 0 ) THEN RETURN; END_IF
// dec remaining parameter(s)                        
ParameterCnt := ParameterCnt - 1;
// Create log entry for Progress
CreateLogMessagePara1 ( Timestamp   := Timestamp,
                        MessageType := MessageType.CMD,
                        Severity    := Severity.DEBUG,
                        MessageCode := 0,
                        MessageText := 'Response.Progress = {1}',
                        Para1       :=  UINT_TO_STRING(_response.Progress));


// Return if no parameter is remaining...
IF ( ParameterCnt = 0 ) THEN RETURN; END_IF
// dec remaining parameter(s)                        
ParameterCnt := ParameterCnt - 1;
// Create log entry for RemainingDistance
CreateLogMessagePara1 ( Timestamp   := Timestamp,
                        MessageType := MessageType.CMD,
                        Severity    := Severity.DEBUG,
                        MessageCode := 0,
                        MessageText := 'Response.RemainingDistance = {1}',
                        Para1       :=  REAL_TO_STRING(_response.RemainingDistance));


// Return if no parameter is remaining...
IF ( ParameterCnt = 0 ) THEN RETURN; END_IF
// dec remaining parameter(s)                        
ParameterCnt := ParameterCnt - 1;
// Create log entry for InClamping
CreateLogMessagePara1 ( Timestamp   := Timestamp,
                        MessageType := MessageType.CMD,
                        Severity    := Severity.DEBUG,
                        MessageCode := 0,
                        MessageText := 'Response.InClamping = {1}',
                        Para1       :=  BOOL_TO_STRING(_response.InClamping));

                
END_METHOD

METHOD PROTECTED Reset : DINT
VAR_INPUT
END_VAR
                  Reset := SUPER^.Reset();

Done               := FALSE;
Busy               := FALSE;
Active             := FALSE;
CommandBuffered    := FALSE;
CommandAborted     := FALSE;
CommandInterrupted := FALSE;


                
END_METHOD
END_FUNCTION_BLOCK

/// Create spline on RC from positions stored in PLC
FUNCTION_BLOCK MC_CreateSplineFB EXTENDS RobotLibraryBaseExecuteFB
// ------------------------------------------------------------------------- 
//  SRCI Robot Library                                                
// ------------------------------------------------------------------------- 
//                                                                           
//  Object:      CreateSplineFB                                       
//  Author:      Thorsten Brach                                                
//  Date:        2024-06-01
//
//  Description:                                              
//   
//                                                                           
//  Copyright: 
//    (C) 2024 Thorsten Brach. All rights reserved                                                                                                                                            
//             Licensed under the MIT License.
//                                                                           
//  Disclaimer:                                                                           
//    This project is provided without any guarantee and can be used for   
//    private and commercial purposes. Any use is at the user’s 
//    own risk and responsibility.
//
// -------------------------------------------------------------------------
VAR_INPUT
  /// command parameter 
  ParCmd          : CreateSplineParCmd;
END_VAR
VAR_OUTPUT
  /// Command is transferred and confirmed by the RC
  CommandBuffered : BOOL;
  /// command results
  OutCmd          : CreateSplineOutCmd;     
END_VAR

VAR
  /// internal copy of command parameter 
 _parCmd          : CreateSplineParCmd;
  /// command data to send
 _command         : CreateSplineSendData;
  /// response data received
 _response        : CreateSplineRecvData;      
END_VAR

            SUPER^(AxesGroup := AxesGroup);
          

METHOD INTERNAL CheckAddParameter : BOOL
VAR_INPUT
  /// Payload pointer
  PayloadPtr : UDINT;
END_VAR
VAR
  /// Payload as byte array
  Payload    : ARRAY [1..SIZEOF(_command)] OF BYTE;
  /// Null Byte array 
  Null       : ARRAY [1..SIZEOF(_command)] OF BYTE;
  /// Data length to compare
  DataLen    : UDINT;
END_VAR
                  // Payload pointer must be decreased by one byte, because ADR(Payload) is already one byte !
PayloadPtr := LIMIT (0, PayloadPtr - 1, SIZEOF(Payload) -1);
// Convert command struct to payload array
SysDepMemCpy( pDest := ADR(Payload), pSrc := ADR(_command), DataLen := SIZEOF(_command));
// Calculate the data length to compare - at least one byte must be compared !
DataLen := LIMIT(1, SIZEOF(Payload) - PayloadPtr, SIZEOF(Payload)); 
// Compare Payload-Array with Null-Byte-Array
CheckAddParameter := SysDepMemCmp( pData1 := ADR(Payload) + PayloadPtr , pData2 := ADR(Null), DataLen := DataLen) <>  RobotLibraryConstants.OK ;
                
END_METHOD

METHOD PROTECTED CheckFunctionSupported : BOOL
VAR_IN_OUT
  /// Robot assignment of function
  AxesGroup : AxesGroup; 
END_VAR
                  CheckFunctionSupported := AxesGroup.State.RobotData.RCSupportedFunctions.CreateSpline;

IF ( NOT CheckFunctionSupported )
THEN
  // call base implementation for set error and create log entry
  SUPER^.CheckFunctionSupported(AxesGroup := AxesGroup);
END_IF
                
END_METHOD

METHOD PROTECTED CheckParameterChanged : BOOL
VAR_IN_OUT
  /// Robot assignment of function
  AxesGroup    : AxesGroup; 
END_VAR
                  // Check ParCmd Size is > 0, because MemCmp does not work correctly with size = 0
IF (SIZEOF(ParCmd) = 0) OR (_stepCmd = 0)
THEN 
  RETURN;
END_IF

// compare memory 
_parameterChanged := ( SysDepMemCmp(pData1 := ADR(ParCmd), pData2 := ADR(_parCmd), DataLen := SIZEOF(ParCmd)) <> RobotLibraryConstants.OK );

// check parameter valid ?
_parameterValid   := CheckParameterValid( AxesGroup := AxesGroup );

IF ((  _parameterChanged        )  AND 
    (  _parameterValid          )) OR
    (  _parameterUpdateInternal )  
THEN  
  // Create log entry for parameter changed event
  CreateLogMessagePara1 ( Timestamp   := AxesGroup.State.SystemTime,
                          MessageType := MessageType.CMD,
                          Severity    := Severity.DEBUG,
                          MessageCode := 0,
                          MessageText := 'NotifyParameterChanged Event {1}',
                          Para1       :=  '' );

  // reset internal flag for send parameter update
 _parameterUpdateInternal := FALSE;
  // update internal copy of parameters 
 _parCmd := ParCmd;
  // inc parameter sequence
 _command.ParSeq := _command.ParSeq + 1;
  // update command data  
  CommandData := CreateCommandPayload(AxesGroup := AxesGroup); // ( Access via reference to rCommandFB in ACR )
  // notify active command register 
  AxesGroup.Acyclic.ActiveCommandRegister.NotifyParameterChanged := _uniqueID;
END_IF
                
END_METHOD

METHOD PROTECTED CheckParameterValid : BOOL
VAR_IN_OUT
  /// Robot assignment of function
  AxesGroup : AxesGroup; 
END_VAR
VAR
  /// internal index for loops
 _idx : DINT;
END_VAR
                  CheckParameterValid := TRUE;


// Check ParCmd.Mode valid ? 
IF (( ParCmd.Mode <> SplineMode.DISCRETE_POINTS      ) AND
    ( ParCmd.Mode <> SplineMode.BEZIER_SPLINE        ) AND 
    ( ParCmd.Mode <> SplineMode.B_SPLINES            ) AND 
    ( ParCmd.Mode <> SplineMode.CUBIC_HERMITE_SPLINE ) AND 
    ( ParCmd.Mode <> SplineMode.C_SPLINES    ))  
THEN
  // Parameter not valid
  CheckParameterValid := FALSE;
  // Set error
  SetError( ErrorID := RobotLibraryErrorIdEnum.ERR_INVALID_PAR_CMD, Overwrite := TRUE );
  // Create log entry
  CreateLogMessagePara1 ( Timestamp   := AxesGroup.State.SystemTime,
                          MessageType := MessageType.CMD,
                          Severity    := Severity.ERROR,
                          MessageCode := ErrorID,
                          MessageText := 'Invalid Parameter ParCmd.Mode = {1}',
                          Para1       := SPLINE_MODE_TO_STRING(ParCmd.Mode));
  RETURN;                          
END_IF

FOR _idx := 0 TO RobotLibraryParameter.SPLINE_DATA_MAX
DO
  // Check ParCmd.SplineData[x].Position.X valid ? 
  IF ( SysDepIsValidReal(ParCmd.SplineData[_idx].Position.X) = FALSE ) 
  THEN
    // Parameter not valid
    CheckParameterValid := FALSE;
    // Set error
    SetError( ErrorID := RobotLibraryErrorIdEnum.ERR_INVALID_PAR_CMD, Overwrite := TRUE );
    
    // Create log entry
    CreateLogMessagePara2 ( Timestamp   := AxesGroup.State.SystemTime,
                            MessageType := MessageType.CMD,
                            Severity    := Severity.ERROR,
                            MessageCode := ErrorID,
                            MessageText := 'Invalid Parameter ParCmd.[{2}].Position.X = {1}',
                            Para1       := VALID_REAL_TO_STRING(ParCmd.SplineData[_idx].Position.X),
                            Para2       := DINT_TO_STRING(_idx));
    EXIT;                            
    RETURN;                          
  END_IF
  
  
  // Check ParCmd.SplineData[x].Position.Y valid ? 
  IF ( SysDepIsValidReal(ParCmd.SplineData[_idx].Position.Y) = FALSE ) 
  THEN
    // Parameter not valid
    CheckParameterValid := FALSE;
    // Set error
    SetError( ErrorID := RobotLibraryErrorIdEnum.ERR_INVALID_PAR_CMD, Overwrite := TRUE );
    
    // Create log entry
    CreateLogMessagePara2 ( Timestamp   := AxesGroup.State.SystemTime,
                            MessageType := MessageType.CMD,
                            Severity    := Severity.ERROR,
                            MessageCode := ErrorID,
                            MessageText := 'Invalid Parameter ParCmd.SplineData[{2}].Position.Y = {1}',
                            Para1       := VALID_REAL_TO_STRING(ParCmd.SplineData[_idx].Position.Y),
                            Para2       := DINT_TO_STRING(_idx)); 
    EXIT;                            
    RETURN;                          
  END_IF
  
  
  // Check ParCmd.SplineData[x].Position.Z valid ? 
  IF ( SysDepIsValidReal(ParCmd.SplineData[_idx].Position.Z) = FALSE ) 
  THEN
    // Parameter not valid
    CheckParameterValid := FALSE;
    // Set error
    SetError( ErrorID := RobotLibraryErrorIdEnum.ERR_INVALID_PAR_CMD, Overwrite := TRUE );
    
    // Create log entry
    CreateLogMessagePara1 ( Timestamp   := AxesGroup.State.SystemTime,
                            MessageType := MessageType.CMD,
                            Severity    := Severity.ERROR,
                            MessageCode := ErrorID,
                            MessageText := 'Invalid Parameter ParCmd.SplineData[{2}].Position.Z = {1}',
                            Para1       := VALID_REAL_TO_STRING(ParCmd.SplineData[_idx].Position.Z));
    EXIT;                            
    RETURN;                          
  END_IF
  
  
  // Check ParCmd.SplineData[x].Position.Rx valid ? 
  IF ( SysDepIsValidReal(ParCmd.SplineData[_idx].Position.Rx) = FALSE ) 
  THEN
    // Parameter not valid
    CheckParameterValid := FALSE;
    // Set error
    SetError( ErrorID := RobotLibraryErrorIdEnum.ERR_INVALID_PAR_CMD, Overwrite := TRUE );
    
    // Create log entry
    CreateLogMessagePara2 ( Timestamp   := AxesGroup.State.SystemTime,
                            MessageType := MessageType.CMD,
                            Severity    := Severity.ERROR,
                            MessageCode := ErrorID,
                            MessageText := 'Invalid Parameter ParCmd.SplineData[{2}].Position.Rx = {1}',
                            Para1       := VALID_REAL_TO_STRING(ParCmd.SplineData[_idx].Position.Rx),
                            Para2       := DINT_TO_STRING(_idx)); 
    EXIT;                            
    RETURN;                          
  END_IF
  
  
  // Check ParCmd.SplineData[x].Position.Ry valid ? 
  IF ( SysDepIsValidReal(ParCmd.SplineData[_idx].Position.Ry) = FALSE ) 
  THEN
    // Parameter not valid
    CheckParameterValid := FALSE;
    // Set error
    SetError( ErrorID := RobotLibraryErrorIdEnum.ERR_INVALID_PAR_CMD, Overwrite := TRUE );
    
    // Create log entry
    CreateLogMessagePara2 ( Timestamp   := AxesGroup.State.SystemTime,
                            MessageType := MessageType.CMD,
                            Severity    := Severity.ERROR,
                            MessageCode := ErrorID,
                            MessageText := 'Invalid Parameter ParCmd.SplineData[{2}].Position.Ry = {1}',
                            Para1       := VALID_REAL_TO_STRING(ParCmd.SplineData[_idx].Position.Ry),
                            Para2       := DINT_TO_STRING(_idx));
    EXIT;                            
    RETURN;                          
  END_IF
  
  
  // Check ParCmd.SplineData[x].Position.Rz valid ? 
  IF ( SysDepIsValidReal(ParCmd.SplineData[_idx].Position.Rz) = FALSE ) 
  THEN
    // Parameter not valid
    CheckParameterValid := FALSE;
    // Set error
    SetError( ErrorID := RobotLibraryErrorIdEnum.ERR_INVALID_PAR_CMD, Overwrite := TRUE );
    
    // Create log entry
    CreateLogMessagePara2 ( Timestamp   := AxesGroup.State.SystemTime,
                            MessageType := MessageType.CMD,
                            Severity    := Severity.ERROR,
                            MessageCode := ErrorID,
                            MessageText := 'Invalid Parameter ParCmd.SplineData[{2}].Position.Rz = {1}',
                            Para1       := VALID_REAL_TO_STRING(ParCmd.SplineData[_idx].Position.Rz),
                            Para2       := DINT_TO_STRING(_idx));
    EXIT;                            
    RETURN;                          
  END_IF
  
  
  // Check ParCmd.SplineData[x].Position.E1 valid ? 
  IF ( SysDepIsValidReal(ParCmd.SplineData[_idx].Position.E1) = FALSE ) 
  THEN
    // Parameter not valid
    CheckParameterValid := FALSE;
    // Set error
    SetError( ErrorID := RobotLibraryErrorIdEnum.ERR_INVALID_PAR_CMD, Overwrite := TRUE );
    
    // Create log entry
    CreateLogMessagePara2 ( Timestamp   := AxesGroup.State.SystemTime,
                            MessageType := MessageType.CMD,
                            Severity    := Severity.ERROR,
                            MessageCode := ErrorID,
                            MessageText := 'Invalid Parameter ParCmd.SplineData[{2}].Position.E1 = {1}',
                            Para1       := VALID_REAL_TO_STRING(ParCmd.SplineData[_idx].Position.E1),
                            Para2       := DINT_TO_STRING(_idx));
    EXIT;                            
    RETURN;                          
  END_IF
  
  
  // Check ParCmd.SplineData[x].Position.E2 valid ? 
  IF ( SysDepIsValidReal(ParCmd.SplineData[_idx].Position.E2) = FALSE ) 
  THEN
    // Parameter not valid
    CheckParameterValid := FALSE;
    // Set error
    SetError( ErrorID := RobotLibraryErrorIdEnum.ERR_INVALID_PAR_CMD, Overwrite := TRUE );
    
    // Create log entry
    CreateLogMessagePara2 ( Timestamp   := AxesGroup.State.SystemTime,
                            MessageType := MessageType.CMD,
                            Severity    := Severity.ERROR,
                            MessageCode := ErrorID,
                            MessageText := 'Invalid Parameter ParCmd.SplineData[{2}].Position.E2 = {1}',
                            Para1       := VALID_REAL_TO_STRING(ParCmd.SplineData[_idx].Position.E2),
                            Para2       := DINT_TO_STRING(_idx)); 
    EXIT;                            
    RETURN;                          
  END_IF
  
  
  // Check ParCmd.SplineData[_idx].Position.E3 valid ? 
  IF ( SysDepIsValidReal(ParCmd.SplineData[_idx].Position.E3) = FALSE ) 
  THEN
    // Parameter not valid
    CheckParameterValid := FALSE;
    // Set error
    SetError( ErrorID := RobotLibraryErrorIdEnum.ERR_INVALID_PAR_CMD, Overwrite := TRUE );
    
    // Create log entry
    CreateLogMessagePara2 ( Timestamp   := AxesGroup.State.SystemTime,
                            MessageType := MessageType.CMD,
                            Severity    := Severity.ERROR,
                            MessageCode := ErrorID,
                            MessageText := 'Invalid Parameter ParCmd.SplineData[{2}].Position.E3 = {1}',
                            Para1       := VALID_REAL_TO_STRING(ParCmd.SplineData[_idx].Position.E3),
                            Para2       := DINT_TO_STRING(_idx));
    EXIT;                            
    RETURN;                          
  END_IF
  
  
  // Check ParCmd.SplineData[x].Position.E4 valid ? 
  IF ( SysDepIsValidReal(ParCmd.SplineData[_idx].Position.E4) = FALSE ) 
  THEN
    // Parameter not valid
    CheckParameterValid := FALSE;
    // Set error
    SetError( ErrorID := RobotLibraryErrorIdEnum.ERR_INVALID_PAR_CMD, Overwrite := TRUE );
    
    // Create log entry
    CreateLogMessagePara2 ( Timestamp   := AxesGroup.State.SystemTime,
                            MessageType := MessageType.CMD,
                            Severity    := Severity.ERROR,
                            MessageCode := ErrorID,
                            MessageText := 'Invalid Parameter ParCmd.SplineData[{2}].Position.E4 = {1}',
                            Para1       := VALID_REAL_TO_STRING(ParCmd.SplineData[_idx].Position.E4),
                            Para2       := DINT_TO_STRING(_idx));
    EXIT;                            
    RETURN;                          
  END_IF
  
  
  // Check ParCmd.SplineData[x].Position.E5 valid ? 
  IF ( SysDepIsValidReal(ParCmd.SplineData[_idx].Position.E5) = FALSE ) 
  THEN
    // Parameter not valid
    CheckParameterValid := FALSE;
    // Set error
    SetError( ErrorID := RobotLibraryErrorIdEnum.ERR_INVALID_PAR_CMD, Overwrite := TRUE );
    
    // Create log entry
    CreateLogMessagePara2 ( Timestamp   := AxesGroup.State.SystemTime,
                            MessageType := MessageType.CMD,
                            Severity    := Severity.ERROR,
                            MessageCode := ErrorID,
                            MessageText := 'Invalid Parameter ParCmd.SplineData[{2}].Position.E5 = {1}',
                            Para1       := VALID_REAL_TO_STRING(ParCmd.SplineData[_idx].Position.E5),
                            Para2       := DINT_TO_STRING(_idx));
    EXIT;                            
    RETURN;                          
  END_IF
  
  
  // Check ParCmd.SplineData[x].Position.E6 valid ? 
  IF ( SysDepIsValidReal(ParCmd.SplineData[_idx].Position.E6) = FALSE ) 
  THEN
    // Parameter not valid
    CheckParameterValid := FALSE;
    // Set error
    SetError( ErrorID := RobotLibraryErrorIdEnum.ERR_INVALID_PAR_CMD, Overwrite := TRUE );
    
    // Create log entry
    CreateLogMessagePara2 ( Timestamp   := AxesGroup.State.SystemTime,
                            MessageType := MessageType.CMD,
                            Severity    := Severity.ERROR,
                            MessageCode := ErrorID,
                            MessageText := 'Invalid Parameter ParCmd.SplineData[{2}].Position.E6 = {1}',
                            Para1       := VALID_REAL_TO_STRING(ParCmd.SplineData[_idx].Position.E6),
                            Para2       := DINT_TO_STRING(_idx));
    EXIT;                            
    RETURN;                          
  END_IF
  
  
  // Check ParCmd.SplineData[x].Position.Config.Shoulder valid ? 
  IF (( ParCmd.SplineData[_idx].Position.Config.Shoulder <> ArmConfigShoulder.USE_CONFIG ) AND  
      ( ParCmd.SplineData[_idx].Position.Config.Shoulder <> ArmConfigShoulder.SAME       ) AND
      ( ParCmd.SplineData[_idx].Position.Config.Shoulder <> ArmConfigShoulder.FREE       ) AND
      ( ParCmd.SplineData[_idx].Position.Config.Shoulder <> ArmConfigShoulder.BACK       ) AND
      ( ParCmd.SplineData[_idx].Position.Config.Shoulder <> ArmConfigShoulder.FRONT      ))
  THEN
    // Parameter not valid
    CheckParameterValid := FALSE;
    // Set error
    SetError( ErrorID := RobotLibraryErrorIdEnum.ERR_CONFIGMODE_SHOULDER_INVALID, Overwrite := TRUE );
    // Create log entry
    CreateLogMessagePara2 ( Timestamp   := AxesGroup.State.SystemTime,
                            MessageType := MessageType.CMD,
                            Severity    := Severity.ERROR,
                            MessageCode := ErrorID,
                            MessageText := 'Invalid Parameter ParCmd.SplineData[{2}].Position.Config.Shoulder = {1}',
                            Para1       := ARM_CONFIG_SHOULDER_TO_STRING(ParCmd.SplineData[_idx].Position.Config.Shoulder),
                            Para2       := DINT_TO_STRING(_idx));
    EXIT;                            
    RETURN;                          
  END_IF
  
  
  // Check ParCmd.SplineData[x].Position.Config.Elbow valid ? 
  IF (( ParCmd.SplineData[_idx].Position.Config.Elbow <> ArmConfigElbow.USE_CONFIG ) AND  
      ( ParCmd.SplineData[_idx].Position.Config.Elbow <> ArmConfigElbow.SAME       ) AND
      ( ParCmd.SplineData[_idx].Position.Config.Elbow <> ArmConfigElbow.FREE       ) AND
      ( ParCmd.SplineData[_idx].Position.Config.Elbow <> ArmConfigElbow.DOWN       ) AND
      ( ParCmd.SplineData[_idx].Position.Config.Elbow <> ArmConfigElbow.UP         ))
  THEN
    // Parameter not valid
    CheckParameterValid := FALSE;
    // Set error
    SetError( ErrorID := RobotLibraryErrorIdEnum.ERR_CONFIGMODE_ELBOW_INVALID, Overwrite := TRUE );
    // Create log entry
    CreateLogMessagePara2 ( Timestamp   := AxesGroup.State.SystemTime,
                            MessageType := MessageType.CMD,
                            Severity    := Severity.ERROR,
                            MessageCode := ErrorID,
                            MessageText := 'Invalid Parameter ParCmd.SplineData[{2}].Position.Config.Elbow = {1}',
                            Para1       := ARM_CONFIG_ELBOW_TO_STRING(ParCmd.SplineData[_idx].Position.Config.Elbow),
                            Para2       := DINT_TO_STRING(_idx));
    EXIT;                            
    RETURN;                          
  END_IF
  
  
  // Check ParCmd.SplineData[x].Position.Config.Wrist valid ? 
  IF (( ParCmd.SplineData[_idx].Position.Config.Wrist <> ArmConfigWrist.USE_CONFIG ) AND  
      ( ParCmd.SplineData[_idx].Position.Config.Wrist <> ArmConfigWrist.SAME       ) AND
      ( ParCmd.SplineData[_idx].Position.Config.Wrist <> ArmConfigWrist.FREE       ) AND
      ( ParCmd.SplineData[_idx].Position.Config.Wrist <> ArmConfigWrist.FLIP       ) AND
      ( ParCmd.SplineData[_idx].Position.Config.Wrist <> ArmConfigWrist.NON_FLIP   ))
  THEN
    // Parameter not valid
    CheckParameterValid := FALSE;
    // Set error
    SetError( ErrorID := RobotLibraryErrorIdEnum.ERR_CONFIGMODE_WRIST_INVALID, Overwrite := TRUE );
    // Create log entry
    CreateLogMessagePara2 ( Timestamp   := AxesGroup.State.SystemTime,
                            MessageType := MessageType.CMD,
                            Severity    := Severity.ERROR,
                            MessageCode := ErrorID,
                            MessageText := 'Invalid Parameter ParCmd.SplineData[{2}].Position.Config.Wrist = {1}',
                            Para1       := ARM_CONFIG_WRIST_TO_STRING(ParCmd.SplineData[_idx].Position.Config.Wrist),
                            Para2       := DINT_TO_STRING(_idx));      
    EXIT;                            
    RETURN;                          
  END_IF

  
  // Check ParCmd.SplineData[x].VelocityRate valid ? 
  IF  (( SysDepIsValidReal(ParCmd.SplineData[_idx].VelocityRate) = FALSE )  OR
      ((                   ParCmd.SplineData[_idx].VelocityRate  <     0 )  AND 
       (                   ParCmd.SplineData[_idx].VelocityRate <>    -1 )) OR   
       (                   ParCmd.SplineData[_idx].VelocityRate  >   100 ))      
  THEN
    // Parameter not valid
    CheckParameterValid := FALSE;
    // Set error
    SetError( ErrorID := RobotLibraryErrorIdEnum.ERR_VELOCITY_INVALID, Overwrite := TRUE );
    // Create log entry
    CreateLogMessagePara2 ( Timestamp   := AxesGroup.State.SystemTime,
                            MessageType := MessageType.CMD,
                            Severity    := Severity.ERROR,
                            MessageCode := ErrorID,
                            MessageText := 'Invalid Parameter ParCmd.SplineData[{2}].VelocityRate = {1}',
                            Para1       := VALID_REAL_TO_STRING(ParCmd.SplineData[_idx].VelocityRate),
                            Para2       := DINT_TO_STRING(_idx));                            
    EXIT;                            
    RETURN;
  END_IF
  
  
  // Check ParCmd.SplineData[x].AccelerationRate valid ? 
  IF  (( SysDepIsValidReal(ParCmd.SplineData[_idx].AccelerationRate) = FALSE )  OR
      ((                   ParCmd.SplineData[_idx].AccelerationRate  <     0 )  AND 
       (                   ParCmd.SplineData[_idx].AccelerationRate <>    -1 )) OR   
       (                   ParCmd.SplineData[_idx].AccelerationRate  >   100 ))      
  THEN
    // Parameter not valid
    CheckParameterValid := FALSE;
    // Set error
    SetError( ErrorID := RobotLibraryErrorIdEnum.ERR_ACCELERATION_INVALID, Overwrite := TRUE );
    // Create log entry
    CreateLogMessagePara2 ( Timestamp   := AxesGroup.State.SystemTime,
                            MessageType := MessageType.CMD,
                            Severity    := Severity.ERROR,
                            MessageCode := ErrorID,
                            MessageText := 'Invalid Parameter ParCmd.SplineData[{2}].AccelerationRate = {1}',
                            Para1       := VALID_REAL_TO_STRING(ParCmd.SplineData[_idx].AccelerationRate),
                            Para2       := DINT_TO_STRING(_idx));
    EXIT;                            
    RETURN;
  END_IF
  
  
  // Check ParCmd.SplineData[x].DecelerationRate valid ? 
  IF  (( SysDepIsValidReal(ParCmd.SplineData[_idx].DecelerationRate) = FALSE )  OR
      ((                   ParCmd.SplineData[_idx].DecelerationRate  <     0 )  AND 
       (                   ParCmd.SplineData[_idx].DecelerationRate <>    -1 )) OR   
       (                   ParCmd.SplineData[_idx].DecelerationRate  >   100 ))      
  THEN
    // Parameter not valid
    CheckParameterValid := FALSE;
    // Set error
    SetError( ErrorID := RobotLibraryErrorIdEnum.ERR_DECELERATION_INVALID, Overwrite := TRUE );
    // Create log entry
    CreateLogMessagePara2 ( Timestamp   := AxesGroup.State.SystemTime,
                            MessageType := MessageType.CMD,
                            Severity    := Severity.ERROR,
                            MessageCode := ErrorID,
                            MessageText := 'Invalid Parameter ParCmd.SplineData[{2}].DecelerationRate = {1}',
                            Para1       := VALID_REAL_TO_STRING(ParCmd.SplineData[_idx].DecelerationRate),
                            Para2       := DINT_TO_STRING(_idx));                            
    EXIT;                            
    RETURN;
  END_IF
  
  
  // Check ParCmd.SplineData[x].JerkRate valid ? 
  IF  (( SysDepIsValidReal(ParCmd.SplineData[_idx].JerkRate) = FALSE )  OR
      ((                   ParCmd.SplineData[_idx].JerkRate  <     0 )  AND 
       (                   ParCmd.SplineData[_idx].JerkRate <>    -1 )) OR   
       (                   ParCmd.SplineData[_idx].JerkRate  >   100 ))      
  THEN
    // Parameter not valid
    CheckParameterValid := FALSE;
    // Set error
    SetError( ErrorID := RobotLibraryErrorIdEnum.ERR_JERK_INVALID, Overwrite := TRUE );
    // Create log entry
    CreateLogMessagePara2 ( Timestamp   := AxesGroup.State.SystemTime,
                            MessageType := MessageType.CMD,
                            Severity    := Severity.ERROR,
                            MessageCode := ErrorID,
                            MessageText := 'Invalid Parameter ParCmd.SplineData[{2}].JerkRate = {1}',
                            Para1       := VALID_REAL_TO_STRING(ParCmd.SplineData[_idx].JerkRate),
                            Para2       := DINT_TO_STRING(_idx));                            
    EXIT;                            
    RETURN;
  END_IF
  
  
  // Check ParCmd.SplineData[x].ToolNo valid ? 
  IF (( ParCmd.SplineData[_idx].ToolNo <   0 ) OR   
      ( ParCmd.SplineData[_idx].ToolNo > 254 ))
  THEN
    // Parameter not valid
    CheckParameterValid := FALSE;
    // Set error
    SetError( ErrorID := RobotLibraryErrorIdEnum.ERR_INVALID_PAR_CMD, Overwrite := TRUE );
    // Create log entry
    CreateLogMessagePara2 ( Timestamp   := AxesGroup.State.SystemTime,
                            MessageType := MessageType.CMD,
                            Severity    := Severity.ERROR,
                            MessageCode := ErrorID,
                            MessageText := 'Invalid Parameter ParCmd.SplineData[{2}].ToolNo = {1}',
                            Para1       := USINT_TO_STRING(ParCmd.SplineData[_idx].ToolNo),
                            Para2       := DINT_TO_STRING(_idx));                           
    EXIT;                            
    RETURN;
  END_IF
  
  
  // Check ParCmd.SplineData[x].FrameNo valid ? 
  IF (( ParCmd.SplineData[_idx].FrameNo <   0 ) OR   
      ( ParCmd.SplineData[_idx].FrameNo > 254 ))
  THEN
    // Parameter not valid
    CheckParameterValid := FALSE;
    // Set error
    SetError( ErrorID := RobotLibraryErrorIdEnum.ERR_INVALID_PAR_CMD, Overwrite := TRUE );
    // Create log entry
    CreateLogMessagePara2 ( Timestamp   := AxesGroup.State.SystemTime,
                            MessageType := MessageType.CMD,
                            Severity    := Severity.ERROR,
                            MessageCode := ErrorID,
                            MessageText := 'Invalid Parameter ParCmd.SplineData[{2}].FrameNo = {1}',
                            Para1       := USINT_TO_STRING(ParCmd.SplineData[_idx].FrameNo),
                            Para2       := DINT_TO_STRING(_idx));                            
    EXIT;                            
    RETURN;
  END_IF

    
  // Check ParCmd.SplineData[x].MoveTime valid ? 
  IF  ( ParCmd.SplineData[_idx].MoveTime < T#0S )
  THEN
    // Parameter not valid
    CheckParameterValid := FALSE;
    // Set error
    SetError( ErrorID := RobotLibraryErrorIdEnum.ERR_INVALID_PAR_CMD, Overwrite := TRUE );
    // Create log entry
    CreateLogMessagePara2 ( Timestamp   := AxesGroup.State.SystemTime,
                            MessageType := MessageType.CMD,
                            Severity    := Severity.ERROR,
                            MessageCode := ErrorID,
                            MessageText := 'Invalid Parameter ParCmd.SplineData[{2}].MoveTime = {1}',
                            Para1       := TIME_TO_STRING(ParCmd.SplineData[_idx].MoveTime),
                            Para2       := DINT_TO_STRING(_idx));                           
    EXIT;                            
    RETURN;
  END_IF  
END_FOR

                
END_METHOD

METHOD INTERNAL CreateCommandPayload : RobotLibraryCommandDataFB
VAR_IN_OUT
  /// Robot assignment of function
  AxesGroup : AxesGroup; 
END_VAR
VAR
  /// Parameter count
 _parameterCnt : DINT;
END_VAR
// Table 6-754: Sent CMD payload (PLC to RC) of "CreateSpline"
// --------------------------
// Header
// --------------------------
// Byte 00 : UINT  - Type HB     
// Byte 01 :       - Type LB    
// Byte 02 : USINT - Reserve | ExecutionMode
// Byte 03 : USINT - ParSeq  | Priority
// --------------------------
// Datablock
// --------------------------
// Byte 04 : UINT  Mode;
// Byte 05 : SINT  SplineID;
// Byte 06 : UINT  SplineData.VelocityRate;
// Byte 07 :       SplineData.VelocityRate;
// Byte 08 : UINT  SplineData.AccelerationRate;
// Byte 09 :       SplineData.AccelerationRate;
// Byte 10 : UINT  SplineData.DecelerationRate;
// Byte 11 :       SplineData.DecelerationRate;
// Byte 12 : UINT  SplineData.JerkRate;
// Byte 13 :       SplineData.JerkRate;
// Byte 14 : USINT SplineData.ToolNo;
// Byte 15 : USINT SplineData.FrameNo;
// Byte 16 : REAL  SplineData.X;
// Byte 17 :       SplineData.X;
// Byte 18 :       SplineData.X;
// Byte 19 :       SplineData.X;
// Byte 20 : REAL  SplineData.Y;
// Byte 21 :       SplineData.Y;
// Byte 22 :       SplineData.Y;
// Byte 23 :       SplineData.Y;
// Byte 24 : REAL  SplineData.Z;
// Byte 25 :       SplineData.Z;
// Byte 26 :       SplineData.Z;
// Byte 27 :       SplineData.Z;
// Byte 28 : REAL  SplineData.RX;
// Byte 29 :       SplineData.RX;
// Byte 30 :       SplineData.RX;
// Byte 31 :       SplineData.RX;
// Byte 32 : REAL  SplineData.RY;
// Byte 33 :       SplineData.RY;
// Byte 34 :       SplineData.RY;
// Byte 35 :       SplineData.RY;
// Byte 36 : REAL  SplineData.RZ;
// Byte 37 :       SplineData.RZ;
// Byte 38 :       SplineData.RZ;
// Byte 39 :       SplineData.RZ;
// Byte 40 : BYTE  - - - - - W E S;
// Byte 41 : BYTE  Reserved;
// Byte 42 : BYTE  SplineData.TurnNumber[0];
// Byte 43 : BYTE  SplineData.TurnNumber[1];
// Byte 44 : BYTE  SplineData.TurnNumber[2];
// Byte 45 : BYTE  SplineData.TurnNumber[3];
// Byte 46 : REAL  SplineData.E1;
// Byte 47 :       SplineData.E1;
// Byte 48 :       SplineData.E1;
// Byte 49 :       SplineData.E1;
// Byte 50 : UINT  SplineData.Time;
// Byte 51 :       SplineData.Time;
// Byte 52 : REAL  SplineData.E2;
// Byte 53 :       SplineData.E2;
// Byte 54 :       SplineData.E2;
// Byte 55 :       SplineData.E2;
// Byte 56 : REAL  SplineData.E3;
// Byte 57 :       SplineData.E3;
// Byte 58 :       SplineData.E3;
// Byte 59 :       SplineData.E3;
// Byte 60 : REAL  SplineData.E4;
// Byte 61 :       SplineData.E4;
// Byte 62 :       SplineData.E4;
// Byte 63 :       SplineData.E4;
// Byte 64 : REAL  SplineData.E5;
// Byte 65 :       SplineData.E5;
// Byte 66 :       SplineData.E5;
// Byte 67 :       SplineData.E5;
// Byte 68 : REAL  SplineData.E6;
// Byte 69 :       SplineData.E6;
// Byte 70 :       SplineData.E6;
// Byte 71 :       SplineData.E6;
VAR
  /// internal index for loops
  _idx : DINT;
END_VAR
                  // set command parameter 
_command.CmdTyp   :=  CmdType.CreateSpline;
_command.ExecMode :=  ExecMode;
_command.ParSeq   := _command.ParSeq;
_command.Priority :=  Priority;
_command.Mode     := _parCmd.Mode;
_command.SplineID := _parCmd.SplineID;

FOR _idx := 1 TO RobotLibraryParameter.SPLINE_DATA_MAX
DO
  _command.SplineData[_idx].VelocityRate     := REAL_TO_PERCENT_UINT(_parCmd.SplineData[_idx].VelocityRate     , IsOptional := FALSE);
  _command.SplineData[_idx].AccelerationRate := REAL_TO_PERCENT_UINT(_parCmd.SplineData[_idx].AccelerationRate , IsOptional := FALSE);
  _command.SplineData[_idx].DecelerationRate := REAL_TO_PERCENT_UINT(_parCmd.SplineData[_idx].DecelerationRate , IsOptional := TRUE );
  _command.SplineData[_idx].JerkRate         := REAL_TO_PERCENT_UINT(_parCmd.SplineData[_idx].JerkRate         , IsOptional := TRUE );
  _command.SplineData[_idx].ToolNo           :=              _parCmd.SplineData[_idx].ToolNo;
  _command.SplineData[_idx].FrameNo          :=              _parCmd.SplineData[_idx].FrameNo;
  _command.SplineData[_idx].MoveTime         := TIME_TO_UINT(_parCmd.SplineData[_idx].MoveTime);
END_FOR

// copy command data to header
_cmdHeader := _command;
// call base implementation to copy header to payload buffer
CreateCommandPayload := SUPER^.CreateCommandPayload(AxesGroup := AxesGroup);


// Check parameter must be added ? 
IF ( CheckAddParameter(CreateCommandPayload.PayloadPtr))
THEN
  // add command.Mode
  CreateCommandPayload.AddUint(_command.Mode);
  // inc parameter counter
 _parameterCnt := _parameterCnt + 1;  
END_IF


// Check parameter must be added ? 
IF ( CheckAddParameter(CreateCommandPayload.PayloadPtr))
THEN
  // add command.SplineID
  CreateCommandPayload.AddSint(_command.SplineID);
  // inc parameter counter
 _parameterCnt := _parameterCnt + 1;  
END_IF


FOR _idx := 1 TO RobotLibraryParameter.SPLINE_DATA_MAX
DO
  // Check parameter must be added ? 
  IF ( CheckAddParameter(CreateCommandPayload.PayloadPtr))
  THEN
    // add command.VelocityRate
    CreateCommandPayload.AddUint(_command.SplineData[_idx].VelocityRate);
    // inc parameter counter
   _parameterCnt := _parameterCnt + 1;  
  END_IF
    
    
  // Check parameter must be added ? 
  IF ( CheckAddParameter(CreateCommandPayload.PayloadPtr))
  THEN
    // add command.AccelerationRate
    CreateCommandPayload.AddUint(_command.SplineData[_idx].AccelerationRate);
    // inc parameter counter
   _parameterCnt := _parameterCnt + 1;  
  END_IF

    
  // Check parameter must be added ? 
  IF ( CheckAddParameter(CreateCommandPayload.PayloadPtr))
  THEN
    // add command.DecelerationRate
    CreateCommandPayload.AddUint(_command.SplineData[_idx].DecelerationRate);
    // inc parameter counter
   _parameterCnt := _parameterCnt + 1;  
  END_IF
  

  // Check parameter must be added ? 
  IF ( CheckAddParameter(CreateCommandPayload.PayloadPtr))
  THEN
    // add command.JerkRate
    CreateCommandPayload.AddUint(_command.SplineData[_idx].JerkRate);
    // inc parameter counter
   _parameterCnt := _parameterCnt + 1;  
  END_IF
  

  // Check parameter must be added ? 
  IF ( CheckAddParameter(CreateCommandPayload.PayloadPtr))
  THEN
    // add command.ToolNo
    CreateCommandPayload.AddUsint(_command.SplineData[_idx].ToolNo);
    // inc parameter counter
   _parameterCnt := _parameterCnt + 1;  
  END_IF
  

  // Check parameter must be added ? 
  IF ( CheckAddParameter(CreateCommandPayload.PayloadPtr))
  THEN
    // add command.FrameNo
    CreateCommandPayload.AddUsint(_command.SplineData[_idx].FrameNo);
    // inc parameter counter
   _parameterCnt := _parameterCnt + 1;  
  END_IF

    
  // Check parameter must be added ? 
  IF ( CheckAddParameter(CreateCommandPayload.PayloadPtr))
  THEN
    // add command.SplineData[_idx].Position.X
    CreateCommandPayload.AddReal(_command.SplineData[_idx].Position.X);
    // inc parameter counter
   _parameterCnt := _parameterCnt + 1;  
  END_IF


  // Check parameter must be added ? 
  IF ( CheckAddParameter(CreateCommandPayload.PayloadPtr))
  THEN
    // add command.SplineData[_idx].Position.Y
    CreateCommandPayload.AddReal(_command.SplineData[_idx].Position.Y);
    // inc parameter counter
   _parameterCnt := _parameterCnt + 1;  
  END_IF
  

  // Check parameter must be added ? 
  IF ( CheckAddParameter(CreateCommandPayload.PayloadPtr))
  THEN
    // add command.SplineData[_idx].Position.Z
    CreateCommandPayload.AddReal(_command.SplineData[_idx].Position.Z);
    // inc parameter counter
   _parameterCnt := _parameterCnt + 1;  
  END_IF
  

  // Check parameter must be added ? 
  IF ( CheckAddParameter(CreateCommandPayload.PayloadPtr))
  THEN
    // add command.SplineData[_idx].Position.Rx
    CreateCommandPayload.AddReal(_command.SplineData[_idx].Position.Rx);
    // inc parameter counter
   _parameterCnt := _parameterCnt + 1;  
  END_IF
  

  // Check parameter must be added ? 
  IF ( CheckAddParameter(CreateCommandPayload.PayloadPtr))
  THEN
    // add command.SplineData[_idx].Position.Ry
    CreateCommandPayload.AddReal(_command.SplineData[_idx].Position.Ry);
    // inc parameter counter
   _parameterCnt := _parameterCnt + 1;  
  END_IF
  

  // Check parameter must be added ? 
  IF ( CheckAddParameter(CreateCommandPayload.PayloadPtr))
  THEN
    // add command.SplineData[_idx].Position.Rz
    CreateCommandPayload.AddReal(_command.SplineData[_idx].Position.Rz);
    // inc parameter counter
   _parameterCnt := _parameterCnt + 1;  
  END_IF
  

  // Check parameter must be added ? 
  IF ( CheckAddParameter(CreateCommandPayload.PayloadPtr))
  THEN
    // add command.SplineData[_idx].Position.Config
    CreateCommandPayload.AddArmConfig(_command.SplineData[_idx].Position.Config);
    // inc parameter counter
   _parameterCnt := _parameterCnt + 1;  
  END_IF
  

  // Check parameter must be added ? 
  IF ( CheckAddParameter(CreateCommandPayload.PayloadPtr))
  THEN
    // add command.SplineData[_idx].Position.TurnNumber
    CreateCommandPayload.AddTurnNumber(_command.SplineData[_idx].Position.TurnNumber);
    // inc parameter counter
   _parameterCnt := _parameterCnt + 1;  
  END_IF
  

  // Check parameter must be added ? 
  IF ( CheckAddParameter(CreateCommandPayload.PayloadPtr))
  THEN
    // add command.SplineData[_idx].Position.E1
    CreateCommandPayload.AddReal(_command.SplineData[_idx].Position.E1);
    // inc parameter counter
   _parameterCnt := _parameterCnt + 1;  
  END_IF
  

  // Check parameter must be added ? 
  IF ( CheckAddParameter(CreateCommandPayload.PayloadPtr))
  THEN
    // add command.SplineData[_idx].MoveTime
    CreateCommandPayload.AddUint(_command.SplineData[_idx].MoveTime);  
    // inc parameter counter
   _parameterCnt := _parameterCnt + 1;  
  END_IF
  

  // Check parameter must be added ? 
  IF ( CheckAddParameter(CreateCommandPayload.PayloadPtr))
  THEN
    // add command.SplineData[_idx].Position.E2
    CreateCommandPayload.AddReal(_command.SplineData[_idx].Position.E2);
    // inc parameter counter
   _parameterCnt := _parameterCnt + 1;  
  END_IF
  

  // Check parameter must be added ? 
  IF ( CheckAddParameter(CreateCommandPayload.PayloadPtr))
  THEN
    // add command.SplineData[_idx].Position.E3
    CreateCommandPayload.AddReal(_command.SplineData[_idx].Position.E3);
    // inc parameter counter
   _parameterCnt := _parameterCnt + 1;  
  END_IF
  

  // Check parameter must be added ? 
  IF ( CheckAddParameter(CreateCommandPayload.PayloadPtr))
  THEN
    // add command.SplineData[_idx].Position.E4
    CreateCommandPayload.AddReal(_command.SplineData[_idx].Position.E4);
    // inc parameter counter
   _parameterCnt := _parameterCnt + 1;  
  END_IF
  

  // Check parameter must be added ? 
  IF ( CheckAddParameter(CreateCommandPayload.PayloadPtr))
  THEN
    // add command.SplineData[_idx].Position.E5
    CreateCommandPayload.AddReal(_command.SplineData[_idx].Position.E5);
    // inc parameter counter
   _parameterCnt := _parameterCnt + 1;  
  END_IF
  

  // Check parameter must be added ? 
  IF ( CheckAddParameter(CreateCommandPayload.PayloadPtr))
  THEN
    // add command.SplineData[_idx].Position.E6
    CreateCommandPayload.AddReal(_command.SplineData[_idx].Position.E6);
    // inc parameter counter
   _parameterCnt := _parameterCnt + 1;  
  END_IF
END_FOR


// Create logging
CreateCommandPayloadLog(AxesGroup := AxesGroup, ParameterCnt := _parameterCnt);
                
END_METHOD

METHOD INTERNAL CreateCommandPayloadLog
VAR_IN_OUT
  /// Robot assignment of function
  AxesGroup : AxesGroup; 
END_VAR
VAR_INPUT
  /// Parameter count
  ParameterCnt : DINT;
END_VAR
VAR 
  /// internal index for loops
 _idx : DINT;
END_VAR
                  // Create log entry for Parameter start
CreateLogMessagePara1 ( Timestamp   := AxesGroup.State.SystemTime,
                        MessageType := MessageType.CMD,
                        Severity    := Severity.DEBUG,
                        MessageCode := 0,
                        MessageText := 'Create command payload with {1} parameter(s) :',
                        Para1       := DINT_TO_STRING(ParameterCnt));


// Return if no parameter is remaining...
IF ( ParameterCnt = 0 ) THEN RETURN; END_IF
// dec remaining parameter(s)                        
ParameterCnt := ParameterCnt - 1;
// Create log entry for Mode
CreateLogMessagePara1 ( Timestamp   := AxesGroup.State.SystemTime,
                        MessageType := MessageType.CMD,
                        Severity    := Severity.DEBUG,
                        MessageCode := 0,
                        MessageText := 'Command.Mode = {1}',
                        Para1       :=  SPLINE_MODE_TO_STRING(_command.Mode));


// Return if no parameter is remaining...
IF ( ParameterCnt = 0 ) THEN RETURN; END_IF
// dec remaining parameter(s)                        
ParameterCnt := ParameterCnt - 1;
// Create log entry for SplineID
CreateLogMessagePara1 ( Timestamp   := AxesGroup.State.SystemTime,
                        MessageType := MessageType.CMD,
                        Severity    := Severity.DEBUG,
                        MessageCode := 0,
                        MessageText := 'Command.SplineID = {1}',
                        Para1       :=  SINT_TO_STRING(_command.SplineID));

// Create log entry for SplineData[x]
FOR _idx := 1 TO RobotLibraryParameter.SPLINE_DATA_MAX
DO
  // Return if no parameter is remaining...
  IF ( ParameterCnt = 0 ) THEN RETURN; END_IF
  // dec remaining parameter(s)                        
  ParameterCnt := ParameterCnt - 1;
  // Create log entry for VelocityRate
  CreateLogMessagePara2 ( Timestamp   := AxesGroup.State.SystemTime,
                          MessageType := MessageType.CMD,
                          Severity    := Severity.DEBUG,
                          MessageCode := 0,
                          MessageText := 'Command.SplineData[{2}].VelocityRate = {1}',
                          Para1       :=  UINT_TO_STRING(_command.SplineData[_idx].VelocityRate),
                          Para2       :=  DINT_TO_STRING(_idx));

                          
  // Return if no parameter is remaining...
  IF ( ParameterCnt = 0 ) THEN RETURN; END_IF
  // dec remaining parameter(s)                        
  ParameterCnt := ParameterCnt - 1;
  // Create log entry for AccelerationRate
  CreateLogMessagePara2 ( Timestamp   := AxesGroup.State.SystemTime,
                          MessageType := MessageType.CMD,
                          Severity    := Severity.DEBUG,
                          MessageCode := 0,
                          MessageText := 'Command.SplineData[{2}].AccelerationRate = {1}',
                          Para1       :=  UINT_TO_STRING(_command.SplineData[_idx].AccelerationRate),
                          Para2       :=  DINT_TO_STRING(_idx));


  // Return if no parameter is remaining...
  IF ( ParameterCnt = 0 ) THEN RETURN; END_IF
  // dec remaining parameter(s)                        
  ParameterCnt := ParameterCnt - 1;
  // Create log entry for DecelerationRate
  CreateLogMessagePara2 ( Timestamp   := AxesGroup.State.SystemTime,
                          MessageType := MessageType.CMD,
                          Severity    := Severity.DEBUG,
                          MessageCode := 0,
                          MessageText := 'Command.SplineData[{2}].DecelerationRate = {1}',
                          Para1       :=  UINT_TO_STRING(_command.SplineData[_idx].DecelerationRate),
                          Para2       :=  DINT_TO_STRING(_idx));
                          

  // Return if no parameter is remaining...
  IF ( ParameterCnt = 0 ) THEN RETURN; END_IF
  // dec remaining parameter(s)                        
  ParameterCnt := ParameterCnt - 1;
  // Create log entry for JerkRate
  CreateLogMessagePara2 ( Timestamp   := AxesGroup.State.SystemTime,
                          MessageType := MessageType.CMD,
                          Severity    := Severity.DEBUG,
                          MessageCode := 0,
                          MessageText := 'Command.SplineData[{2}].JerkRate = {1}',
                          Para1       :=  UINT_TO_STRING(_command.SplineData[_idx].JerkRate),
                          Para2       :=  DINT_TO_STRING(_idx));

                          

  // Return if no parameter is remaining...
  IF ( ParameterCnt = 0 ) THEN RETURN; END_IF
  // dec remaining parameter(s)                        
  ParameterCnt := ParameterCnt - 1;
  // Create log entry for ToolNo
  CreateLogMessagePara2 ( Timestamp   := AxesGroup.State.SystemTime,
                          MessageType := MessageType.CMD,
                          Severity    := Severity.DEBUG,
                          MessageCode := 0,
                          MessageText := 'Command.SplineData[{2}].ToolNo = {1}',
                          Para1       :=  USINT_TO_STRING(_command.SplineData[_idx].ToolNo),
                          Para2       :=  DINT_TO_STRING(_idx));
  

  // Return if no parameter is remaining...
  IF ( ParameterCnt = 0 ) THEN RETURN; END_IF
  // dec remaining parameter(s)                        
  ParameterCnt := ParameterCnt - 1;
  // Create log entry for FrameNo
  CreateLogMessagePara2 ( Timestamp   := AxesGroup.State.SystemTime,
                          MessageType := MessageType.CMD,
                          Severity    := Severity.DEBUG,
                          MessageCode := 0,
                          MessageText := 'Command.SplineData[{2}].FrameNo = {1}',
                          Para1       :=  USINT_TO_STRING(_command.SplineData[_idx].FrameNo),
                          Para2       :=  DINT_TO_STRING(_idx));
                          

  // Return if no parameter is remaining...
  IF ( ParameterCnt = 0 ) THEN RETURN; END_IF
  // dec remaining parameter(s)                        
  ParameterCnt := ParameterCnt - 1;
  // Create log entry for Position.X
  CreateLogMessagePara2 ( Timestamp   := AxesGroup.State.SystemTime,
                          MessageType := MessageType.CMD,
                          Severity    := Severity.DEBUG,
                          MessageCode := 0,
                          MessageText := 'Command.SplineData[{2}].Position.X = {1}',
                          Para1       :=  REAL_TO_STRING(_command.SplineData[_idx].Position.X),
                          Para2       :=  DINT_TO_STRING(_idx));


  // Return if no parameter is remaining...
  IF ( ParameterCnt = 0 ) THEN RETURN; END_IF
  // dec remaining parameter(s)                        
  ParameterCnt := ParameterCnt - 1;
  // Create log entry for Position.Y
  CreateLogMessagePara2 ( Timestamp   := AxesGroup.State.SystemTime,
                          MessageType := MessageType.CMD,
                          Severity    := Severity.DEBUG,
                          MessageCode := 0,
                          MessageText := 'Command.SplineData[{2}].Position.Y = {1}',
                          Para1       :=  REAL_TO_STRING(_command.SplineData[_idx].Position.Y),
                          Para2       :=  DINT_TO_STRING(_idx));
                          

  // Return if no parameter is remaining...
  IF ( ParameterCnt = 0 ) THEN RETURN; END_IF
  // dec remaining parameter(s)                        
  ParameterCnt := ParameterCnt - 1;
  // Create log entry for Position.Z
  CreateLogMessagePara2 ( Timestamp   := AxesGroup.State.SystemTime,
                          MessageType := MessageType.CMD,
                          Severity    := Severity.DEBUG,
                          MessageCode := 0,
                          MessageText := 'Command.SplineData[{2}].Position.Z = {1}',
                          Para1       :=  REAL_TO_STRING(_command.SplineData[_idx].Position.Z),
                          Para2       :=  DINT_TO_STRING(_idx));


  // Return if no parameter is remaining...
  IF ( ParameterCnt = 0 ) THEN RETURN; END_IF
  // dec remaining parameter(s)                        
  ParameterCnt := ParameterCnt - 1;
  // Create log entry for Position.Rx
  CreateLogMessagePara2 ( Timestamp   := AxesGroup.State.SystemTime,
                          MessageType := MessageType.CMD,
                          Severity    := Severity.DEBUG,
                          MessageCode := 0,
                          MessageText := 'Command.SplineData[{2}].Position.Rx = {1}',
                          Para1       :=  REAL_TO_STRING(_command.SplineData[_idx].Position.Rx),
                          Para2       :=  DINT_TO_STRING(_idx));
                          

  // Return if no parameter is remaining...
  IF ( ParameterCnt = 0 ) THEN RETURN; END_IF
  // dec remaining parameter(s)                        
  ParameterCnt := ParameterCnt - 1;
  // Create log entry for Position.Ry
  CreateLogMessagePara2 ( Timestamp   := AxesGroup.State.SystemTime,
                          MessageType := MessageType.CMD,
                          Severity    := Severity.DEBUG,
                          MessageCode := 0,
                          MessageText := 'Command.SplineData[{2}].Position.Ry = {1}',
                          Para1       :=  REAL_TO_STRING(_command.SplineData[_idx].Position.Ry),
                          Para2       :=  DINT_TO_STRING(_idx));
                          

  // Return if no parameter is remaining...
  IF ( ParameterCnt = 0 ) THEN RETURN; END_IF
  // dec remaining parameter(s)                        
  ParameterCnt := ParameterCnt - 1;
  // Create log entry for Position.Rz
  CreateLogMessagePara2 ( Timestamp   := AxesGroup.State.SystemTime,
                          MessageType := MessageType.CMD,
                          Severity    := Severity.DEBUG,
                          MessageCode := 0,
                          MessageText := 'Command.SplineData[{2}].Position.Rz = {1}',
                          Para1       :=  REAL_TO_STRING(_command.SplineData[_idx].Position.Rz),
                          Para2       :=  DINT_TO_STRING(_idx));


  // Return if no parameter is remaining...
  IF ( ParameterCnt = 0 ) THEN RETURN; END_IF
  // dec remaining parameter(s)                        
  ParameterCnt := ParameterCnt - 1;
  // Create log entry for Position.Config
  CreateLogMessagePara2 ( Timestamp   := AxesGroup.State.SystemTime,
                          MessageType := MessageType.CMD,
                          Severity    := Severity.DEBUG,
                          MessageCode := 0,
                          MessageText := 'Command.SplineData[{2}].Position.Config = {1}',
                          Para1       :=  ARM_CONFIG_TO_STRING(_command.SplineData[_idx].Position.Config),
                          Para2       :=  DINT_TO_STRING(_idx));


  // Return if no parameter is remaining...
  IF ( ParameterCnt = 0 ) THEN RETURN; END_IF
  // dec remaining parameter(s)                        
  ParameterCnt := ParameterCnt - 1;
  // Create log entry for Position.TurnNumber[0]
  CreateLogMessagePara2 ( Timestamp   := AxesGroup.State.SystemTime,
                          MessageType := MessageType.CMD,
                          Severity    := Severity.DEBUG,
                          MessageCode := 0,
                          MessageText := 'Command.SplineData[{2}].Position.TurnNumber[0] = {1}',
                          Para1       :=  BYTE_TO_STRING(CombineHalfSints(HalfSintHi := _command.SplineData[_idx].Position.TurnNumber.J2Turns,
                                                                          HalfSintLo := _command.SplineData[_idx].Position.TurnNumber.J1Turns)),                          
                          Para2       :=  DINT_TO_STRING(_idx));


  // Return if no parameter is remaining...
  IF ( ParameterCnt = 0 ) THEN RETURN; END_IF
  // dec remaining parameter(s)                        
  ParameterCnt := ParameterCnt - 1;
  // Create log entry for Position.TurnNumber[1]
  CreateLogMessagePara2 ( Timestamp   := AxesGroup.State.SystemTime,
                          MessageType := MessageType.CMD,
                          Severity    := Severity.DEBUG,
                          MessageCode := 0,
                          MessageText := 'Command.SplineData[{2}].Position.TurnNumber[1] = {1}',
                          Para1       :=  BYTE_TO_STRING(CombineHalfSints(HalfSintHi := _command.SplineData[_idx].Position.TurnNumber.J4Turns,
                                                                          HalfSintLo := _command.SplineData[_idx].Position.TurnNumber.J3Turns)),                          
                          Para2       :=  DINT_TO_STRING(_idx));
                          

  // Return if no parameter is remaining...
  IF ( ParameterCnt = 0 ) THEN RETURN; END_IF
  // dec remaining parameter(s)                        
  ParameterCnt := ParameterCnt - 1;
  // Create log entry for Position.TurnNumber[2]
  CreateLogMessagePara2 ( Timestamp   := AxesGroup.State.SystemTime,
                          MessageType := MessageType.CMD,
                          Severity    := Severity.DEBUG,
                          MessageCode := 0,
                          MessageText := 'Command.SplineData[{2}].Position.TurnNumber[2] = {1}',
                          Para1       :=  BYTE_TO_STRING(CombineHalfSints(HalfSintHi := _command.SplineData[_idx].Position.TurnNumber.J6Turns,
                                                                          HalfSintLo := _command.SplineData[_idx].Position.TurnNumber.J5Turns)),                          
                          Para2       :=  DINT_TO_STRING(_idx));


  // Return if no parameter is remaining...
  IF ( ParameterCnt = 0 ) THEN RETURN; END_IF
  // dec remaining parameter(s)                        
  ParameterCnt := ParameterCnt - 1;
  // Create log entry for Position.TurnNumber[3]
  CreateLogMessagePara2 ( Timestamp   := AxesGroup.State.SystemTime,
                          MessageType := MessageType.CMD,
                          Severity    := Severity.DEBUG,
                          MessageCode := 0,
                          MessageText := 'Command.SplineData[{2}].Position.TurnNumber[3] = {1}',
                          Para1       :=  SINT_TO_STRING(_command.SplineData[_idx].Position.TurnNumber.E1Turns),                          
                          Para2       :=  DINT_TO_STRING(_idx));
                          

  // Return if no parameter is remaining...
  IF ( ParameterCnt = 0 ) THEN RETURN; END_IF
  // dec remaining parameter(s)                        
  ParameterCnt := ParameterCnt - 1;
  // Create log entry for Position.E1
  CreateLogMessagePara2 ( Timestamp   := AxesGroup.State.SystemTime,
                          MessageType := MessageType.CMD,
                          Severity    := Severity.DEBUG,
                          MessageCode := 0,
                          MessageText := 'Command.SplineData[{2}].Position.E1 = {1}',
                          Para1       :=  REAL_TO_STRING(_command.SplineData[_idx].Position.E1),
                          Para2       :=  DINT_TO_STRING(_idx));


  // Return if no parameter is remaining...
  IF ( ParameterCnt = 0 ) THEN RETURN; END_IF
  // dec remaining parameter(s)                        
  ParameterCnt := ParameterCnt - 1;
  // Create log entry for MoveTime
  CreateLogMessagePara2 ( Timestamp   := AxesGroup.State.SystemTime,
                          MessageType := MessageType.CMD,
                          Severity    := Severity.DEBUG,
                          MessageCode := 0,
                          MessageText := 'Command.SplineData[{2}].MoveTime = {1}',
                          Para1       :=  UINT_TO_STRING(_command.SplineData[_idx].MoveTime),
                          Para2       :=  DINT_TO_STRING(_idx));


  // Return if no parameter is remaining...
  IF ( ParameterCnt = 0 ) THEN RETURN; END_IF
  // dec remaining parameter(s)                        
  ParameterCnt := ParameterCnt - 1;
  // Create log entry for Position.E2
  CreateLogMessagePara2 ( Timestamp   := AxesGroup.State.SystemTime,
                          MessageType := MessageType.CMD,
                          Severity    := Severity.DEBUG,
                          MessageCode := 0,
                          MessageText := 'Command.SplineData[{2}].Position.E2 = {1}',
                          Para1       :=  REAL_TO_STRING(_command.SplineData[_idx].Position.E2),
                          Para2       :=  DINT_TO_STRING(_idx));


  // Return if no parameter is remaining...
  IF ( ParameterCnt = 0 ) THEN RETURN; END_IF
  // dec remaining parameter(s)                        
  ParameterCnt := ParameterCnt - 1;
  // Create log entry for Position.E3
  CreateLogMessagePara2 ( Timestamp   := AxesGroup.State.SystemTime,
                          MessageType := MessageType.CMD,
                          Severity    := Severity.DEBUG,
                          MessageCode := 0,
                          MessageText := 'Command.SplineData[{2}].Position.E3 = {1}',
                          Para1       :=  REAL_TO_STRING(_command.SplineData[_idx].Position.E3),
                          Para2       :=  DINT_TO_STRING(_idx));


  // Return if no parameter is remaining...
  IF ( ParameterCnt = 0 ) THEN RETURN; END_IF
  // dec remaining parameter(s)                        
  ParameterCnt := ParameterCnt - 1;
  // Create log entry for Position.E4
  CreateLogMessagePara2 ( Timestamp   := AxesGroup.State.SystemTime,
                          MessageType := MessageType.CMD,
                          Severity    := Severity.DEBUG,
                          MessageCode := 0,
                          MessageText := 'Command.SplineData[{2}].Position.E4 = {1}',
                          Para1       :=  REAL_TO_STRING(_command.SplineData[_idx].Position.E4),
                          Para2       :=  DINT_TO_STRING(_idx));
                          

  // Return if no parameter is remaining...
  IF ( ParameterCnt = 0 ) THEN RETURN; END_IF
  // dec remaining parameter(s)                        
  ParameterCnt := ParameterCnt - 1;
  // Create log entry for Position.E5
  CreateLogMessagePara2 ( Timestamp   := AxesGroup.State.SystemTime,
                          MessageType := MessageType.CMD,
                          Severity    := Severity.DEBUG,
                          MessageCode := 0,
                          MessageText := 'Command.SplineData[{2}].Position.E5 = {1}',
                          Para1       :=  REAL_TO_STRING(_command.SplineData[_idx].Position.E5),
                          Para2       :=  DINT_TO_STRING(_idx));
                          

  // Return if no parameter is remaining...
  IF ( ParameterCnt = 0 ) THEN RETURN; END_IF
  // dec remaining parameter(s)                        
  ParameterCnt := ParameterCnt - 1;
  // Create log entry for Position.E6
  CreateLogMessagePara2 ( Timestamp   := AxesGroup.State.SystemTime,
                          MessageType := MessageType.CMD,
                          Severity    := Severity.DEBUG,
                          MessageCode := 0,
                          MessageText := 'Command.SplineData[{2}].Position.E6 = {1}',
                          Para1       :=  REAL_TO_STRING(_command.SplineData[_idx].Position.E6),
                          Para2       :=  DINT_TO_STRING(_idx));
                          
END_FOR                        
                
END_METHOD

METHOD FB_init : BOOL
VAR_INPUT
  /// if TRUE, the retain variables are initialized (warm start / cold start)
  bInitRetains : BOOL; 
  /// if TRUE, the instance afterwards gets moved into the copy code (online change)
  bInCopyCode  : BOOL;  
END_VAR
                  MyType := 'MC_CreateSplineFB';

ExecMode := ExecutionMode.PARALLEL;
Priority := PriorityLevel.NORMAL;
                
END_METHOD

METHOD PROTECTED OnExecRun : DINT
VAR_IN_OUT
  /// Robot assignment of function
  AxesGroup : AxesGroup; 
END_VAR
                  // call base implementation
SUPER^.OnExecRun(AxesGroup := AxesGroup);

CASE _stepCmd OF
  
  00:  IF ( _execute_R.Q ) AND ( NOT Error)  
       THEN
         // Check function is supported and parameter are valid ?
         IF (( CheckFunctionSupported( AxesGroup := AxesGroup )) AND
             ( CheckParameterValid   ( AxesGroup := AxesGroup )))
         THEN      
           // set busy flag
           Busy := TRUE;
           // Reset command outputs
           SysDepMemSet(pDest := ADR(OutCmd), Value := 0, DataLen := SIZEOF(OutCmd));         
           // apply command parameter
          _parCmd := ParCmd;
           // init parameter sequence
          _command.ParSeq := 1;
           // create command data
           CommandData := CreateCommandPayload(AxesGroup := AxesGroup);
           // Add command to active command register
          _uniqueID := AxesGroup.Acyclic.ActiveCommandRegister.AddCmd( pCommandFB := ADR(THIS^ ));     
           // set timeout
           SetTimeout(PT := _timeoutCmd, rTimer := _timerCmd);
           // inc step counter
          _stepCmd := _stepCmd + 1;
         END_IF 
       END_IF
     

  01:  // Wait for responce received
       IF ( _responseReceived )
       THEN
         // reset response received flag
        _responseReceived := FALSE;
         // update state flags
         OnUpdateStateFlags(_response.State);
         // update state flags
         OnApplyOutCmd(_response.State);
                
         // Done, Aborted or Error ?
         IF (_response.State >= CmdMessageState.DONE )
         THEN
           // set timeout
           SetTimeout(PT := _timeoutCmd, rTimer := _timerCmd);
           // inc step counter
          _stepCmd := _stepCmd + 1; 
         END_IF
       END_IF


  02: IF ( NOT Execute)
      THEN
        Reset(); 
      END_IF     

ELSE
  // invalid step
  SetError( ErrorID := RobotLibraryErrorIdEnum.ERR_INVALID_STEP, Overwrite := TRUE );
END_CASE


// Reset FB
IF ( NOT Execute )
THEN
  Reset();
END_IF
                
END_METHOD

